C01779=-54.382,79.482,17.095,174.9324,20.6601,-3295.6199
C01780=-53.070,81.058,17.237,173.5629,15.1731,-3296.7866
C01781=-52.143,82.495,17.374,174.7815,10.0525,-3297.7041
C01782=-51.202,83.948,17.473,177.1153,6.7838,-3298.6199
C01783=-49.816,85.535,17.521,178.9354,4.2497,-3299.7833
C01784=-47.692,87.339,17.545,179.7213,1.8693,-3301.3630
C01785=-45.077,89.109,17.565,179.9709,0.3614,-3303.1668
C01786=-42.311,90.585,17.585,-179.9996,0.0820,-3304.9634
C01787=-39.610,91.818,17.598,179.9970,0.0075,-3306.6648
C01788=-36.917,92.934,17.598,179.9968,0.0074,-3308.3351
C01789=-34.135,93.972,17.585,179.9985,0.0798,-3310.0366
C01790=-31.135,94.884,17.565,-179.9727,0.3589,-3311.8334
C01791=-28.035,95.481,17.545,-179.7194,1.8706,-3313.6368
C01792=-25.257,95.708,17.521,-178.9370,4.2461,-3315.2169
C01793=-23.155,95.565,17.473,-177.1151,6.7819,-3316.3800
C01794=-21.462,95.203,17.374,-174.7852,10.0480,-3317.2959
C01795=-19.790,94.842,17.237,-173.5645,15.1715,-3318.2136
C01796=-17.748,94.656,17.095,-174.9374,20.6589,-3319.3803
C01797=-14.774,94.777,16.986,-178.0146,24.0591,-3321.1399
C01798=-10.339,95.219,16.941,-179.6989,25.0665,-3323.8030
C01799=-5.406,95.617,16.939,179.9726,25.1250,-3326.7641
C01800=0.000,94.804,18.916,-180.0000,27.0775,-3330.0000
C01801=5.317,94.652,18.914,-179.9702,27.0874,-3333.2152
C01802=10.190,94.262,18.917,179.5911,27.0185,-3336.1699
C01803=14.592,93.857,18.976,177.3137,25.8724,-3338.8371
C01804=17.528,93.824,19.120,173.2655,21.6484,-3340.5819
C01805=19.540,94.146,19.309,171.9611,14.9094,-3341.7253
C01806=21.192,94.676,19.493,173.8561,9.2462,-3342.6169
C01807=22.867,95.222,19.627,176.6046,6.2189,-3343.5035
C01808=24.945,95.538,19.692,178.7208,4.0294,-3344.6333
C01809=27.741,95.446,19.726,179.6779,1.7445,-3346.2063
C01810=30.903,94.927,19.753,179.9766,0.2756,-3348.0324
C01811=33.988,94.020,19.780,179.9962,0.0778,-3349.8748
C01812=36.867,92.953,19.798,-179.9968,0.0074,-3351.6343
C01813=39.659,91.796,19.798,-179.9970,0.0075,-3353.3660
C01814=42.449,90.515,19.780,-179.9981,0.0768,-3355.1253
C01815=45.272,88.975,19.753,-179.9712,0.2718,-3356.9678
C01816=47.874,87.106,19.726,-179.6780,1.7463,-3358.7935
C01817=49.917,85.194,19.692,-178.7206,4.0258,-3360.3670
C01818=51.163,83.502,19.627,-176.6033,6.2165,-3361.4965
C01819=51.961,81.931,19.493,-173.8545,9.2440,-3362.3830
C01820=52.755,80.388,19.309,-171.9613,14.9062,-3363.2751
C01821=53.950,78.738,19.120,-173.2660,21.6521,-3364.4183
C01822=56.048,76.685,18.976,-177.3146,25.8712,-3366.1625
C01823=59.448,73.859,18.917,-179.5906,27.0203,-3368.8301
C01824=63.169,70.689,18.914,179.9644,27.0876,-3371.7846
C01825=67.036,67.036,18.916,-180.0000,27.0793,-3375.0000
C01826=70.689,63.169,18.914,-179.9644,27.0876,-3378.2154
C01827=73.859,59.448,18.917,179.5906,27.0203,-3381.1699
C01828=76.685,56.048,18.976,177.3146,25.8712,-3383.8375
C01829=78.738,53.950,19.120,173.2660,21.6521,-3385.5817
C01830=80.388,52.755,19.309,171.9613,14.9062,-3386.7249
C01831=81.931,51.961,19.493,173.8545,9.2440,-3387.6170
C01832=83.502,51.163,19.627,176.6033,6.2165,-3388.5035
C01833=85.194,49.917,19.692,178.7206,4.0258,-3389.6330
C01834=87.106,47.874,19.726,179.6780,1.7463,-3391.2065
C01835=88.975,45.272,19.753,179.9712,0.2718,-3393.0322
C01836=90.515,42.449,19.780,179.9981,0.0768,-3394.8747
C01837=91.796,39.659,19.798,179.9970,0.0075,-3396.6340
C01838=92.953,36.867,19.798,179.9968,0.0074,-3398.3657
C01839=94.020,33.988,19.780,-179.9962,0.0778,-3400.1252
C01840=94.927,30.903,19.753,-179.9766,0.2756,-3401.9676
C01841=95.446,27.741,19.726,-179.6779,1.7445,-3403.7937
C01842=95.538,24.945,19.692,-178.7208,4.0294,-3405.3667
C01843=95.222,22.867,19.627,-176.6046,6.2189,-3406.4965
C01844=94.676,21.192,19.493,-173.8561,9.2462,-3407.3831
C01845=94.146,19.540,19.309,-171.9611,14.9094,-3408.2747
C01846=93.824,17.528,19.120,-173.2655,21.6484,-3409.4181
C01847=93.857,14.592,18.976,-177.3137,25.8724,-3411.1629
C01848=94.262,10.190,18.917,-179.5911,27.0185,-3413.8301
C01849=94.652,5.317,18.914,179.9702,27.0874,-3416.7848
C01850=94.804,0.000,18.916,180.0000,27.0775,-3420.0000
C01851=94.652,-5.317,18.914,-179.9702,27.0874,-3423.2152
C01852=94.262,-10.190,18.917,179.5911,27.0185,-3426.1699
C01853=93.857,-14.592,18.976,177.3137,25.8724,-3428.8371
C01854=93.824,-17.528,19.120,173.2655,21.6484,-3430.5819
C01855=94.146,-19.540,19.309,171.9611,14.9094,-3431.7253
C01856=94.676,-21.192,19.493,173.8561,9.2462,-3432.6169
C01857=95.222,-22.867,19.627,176.6046,6.2189,-3433.5035
C01858=95.538,-24.945,19.692,178.7208,4.0294,-3434.6333
C01859=95.446,-27.741,19.726,179.6779,1.7445,-3436.2063
C01860=94.927,-30.903,19.753,179.9766,0.2756,-3438.0324
C01861=94.020,-33.988,19.780,179.9962,0.0778,-3439.8748
C01862=92.953,-36.867,19.798,-179.9968,0.0074,-3441.6343
C01863=91.796,-39.659,19.798,-179.9970,0.0075,-3443.3660
C01864=90.515,-42.449,19.780,-179.9981,0.0768,-3445.1253
C01865=88.975,-45.272,19.753,-179.9712,0.2718,-3446.9678
C01866=87.106,-47.874,19.726,-179.6780,1.7463,-3448.7935
C01867=85.194,-49.917,19.692,-178.7206,4.0258,-3450.3670
C01868=83.502,-51.163,19.627,-176.6033,6.2165,-3451.4965
C01869=81.931,-51.961,19.493,-173.8545,9.2440,-3452.3830
C01870=80.388,-52.755,19.309,-171.9613,14.9062,-3453.2751
C01871=78.738,-53.950,19.120,-173.2660,21.6521,-3454.4183
C01872=76.685,-56.048,18.976,-177.3146,25.8712,-3456.1625
C01873=73.859,-59.448,18.917,-179.5906,27.0203,-3458.8301
C01874=70.689,-63.169,18.914,179.9644,27.0876,-3461.7846
C01875=67.036,-67.036,18.916,-180.0000,27.0793,-3465.0000
C01876=63.169,-70.689,18.914,-179.9644,27.0876,-3468.2154
C01877=59.448,-73.859,18.917,179.5906,27.0203,-3471.1699
C01878=56.048,-76.685,18.976,177.3146,25.8712,-3473.8375
C01879=53.950,-78.738,19.120,173.2660,21.6521,-3475.5817
C01880=52.755,-80.388,19.309,171.9613,14.9062,-3476.7249
C01881=51.961,-81.931,19.493,173.8545,9.2440,-3477.6170
C01882=51.163,-83.502,19.627,176.6033,6.2165,-3478.5035
C01883=49.917,-85.194,19.692,178.7206,4.0258,-3479.6330
C01884=47.874,-87.106,19.726,179.6780,1.7463,-3481.2065
C01885=45.272,-88.975,19.753,179.9712,0.2718,-3483.0322
C01886=42.449,-90.515,19.780,179.9981,0.0768,-3484.8747
C01887=39.659,-91.796,19.798,179.9970,0.0075,-3486.6340
C01888=36.867,-92.953,19.798,179.9968,0.0074,-3488.3657
C01889=33.988,-94.020,19.780,-179.9962,0.0778,-3490.1252
C01890=30.903,-94.927,19.753,-179.9766,0.2756,-3491.9676
C01891=27.741,-95.446,19.726,-179.6779,1.7445,-3493.7937
C01892=24.945,-95.538,19.692,-178.7208,4.0294,-3495.3667
C01893=22.867,-95.222,19.627,-176.6046,6.2189,-3496.4965
C01894=21.192,-94.676,19.493,-173.8561,9.2462,-3497.3831
C01895=19.540,-94.146,19.309,-171.9611,14.9094,-3498.2747
C01896=17.528,-93.824,19.120,-173.2655,21.6484,-3499.4181
C01897=14.592,-93.857,18.976,-177.3137,25.8724,-3501.1629
C01898=10.190,-94.262,18.917,-179.5911,27.0185,-3503.8301
C01899=5.317,-94.652,18.914,179.9702,27.0874,-3506.7848
C01900=0.000,-94.804,18.916,-180.0000,27.0775,-3510.0000
C01901=-5.317,-94.652,18.914,-179.9702,27.0874,-3513.2152
C01902=-10.190,-94.262,18.917,179.5911,27.0185,-3516.1699
C01903=-14.592,-93.857,18.976,177.3137,25.8724,-3518.8371
C01904=-17.528,-93.824,19.120,173.2655,21.6484,-3520.5819
C01905=-19.540,-94.146,19.309,171.9611,14.9094,-3521.7253
C01906=-21.192,-94.676,19.493,173.8561,9.2462,-3522.6169
C01907=-22.867,-95.222,19.627,176.6046,6.2189,-3523.5035
C01908=-24.945,-95.538,19.692,178.7208,4.0294,-3524.6333
C01909=-27.741,-95.446,19.726,179.6779,1.7445,-3526.2063
C01910=-30.903,-94.927,19.753,179.9766,0.2756,-3528.0324
C01911=-33.988,-94.020,19.780,179.9962,0.0778,-3529.8748
C01912=-36.867,-92.953,19.798,-179.9968,0.0074,-3531.6343
C01913=-39.659,-91.796,19.798,-179.9970,0.0075,-3533.3660
C01914=-42.449,-90.515,19.780,-179.9981,0.0768,-3535.1253
C01915=-45.272,-88.975,19.753,-179.9712,0.2718,-3536.9678
C01916=-47.874,-87.106,19.726,-179.6780,1.7463,-3538.7935
C01917=-49.917,-85.194,19.692,-178.7206,4.0258,-3540.3670
C01918=-51.163,-83.502,19.627,-176.6033,6.2165,-3541.4965
C01919=-51.961,-81.931,19.493,-173.8545,9.2440,-3542.3830
C01920=-52.755,-80.388,19.309,-171.9613,14.9062,-3543.2751
C01921=-53.950,-78.738,19.120,-173.2660,21.6521,-3544.4183
C01922=-56.048,-76.685,18.976,-177.3146,25.8712,-3546.1625
C01923=-59.448,-73.859,18.917,-179.5906,27.0203,-3548.8301
C01924=-63.169,-70.689,18.914,179.9644,27.0876,-3551.7846
C01925=-67.036,-67.036,18.916,180.0000,27.0793,-3555.0000
C01926=-70.689,-63.169,18.914,-179.9644,27.0876,-3558.2154
C01927=-73.859,-59.448,18.917,179.5906,27.0203,-3561.1699
C01928=-76.685,-56.048,18.976,177.3146,25.8712,-3563.8375
C01929=-78.738,-53.950,19.120,173.2660,21.6521,-3565.5817
C01930=-80.388,-52.755,19.309,171.9613,14.9062,-3566.7249
C01931=-81.931,-51.961,19.493,173.8545,9.2440,-3567.6170
C01932=-83.502,-51.163,19.627,176.6033,6.2165,-3568.5035
C01933=-85.194,-49.917,19.692,178.7206,4.0258,-3569.6330
C01934=-87.106,-47.874,19.726,179.6780,1.7463,-3571.2065
C01935=-88.975,-45.272,19.753,179.9712,0.2718,-3573.0322
C01936=-90.515,-42.449,19.780,179.9981,0.0768,-3574.8747
C01937=-91.796,-39.659,19.798,179.9970,0.0075,-3576.6340
C01938=-92.953,-36.867,19.798,179.9968,0.0074,-3578.3657
C01939=-94.020,-33.988,19.780,-179.9962,0.0778,-3580.1252
C01940=-94.927,-30.903,19.753,-179.9766,0.2756,-3581.9676
C01941=-95.446,-27.741,19.726,-179.6779,1.7445,-3583.7937
C01942=-95.538,-24.945,19.692,-178.7208,4.0294,-3585.3667
C01943=-95.222,-22.867,19.627,-176.6046,6.2189,-3586.4965
C01944=-94.676,-21.192,19.493,-173.8561,9.2462,-3587.3831
C01945=-94.146,-19.540,19.309,-171.9611,14.9094,-3588.2747
C01946=-93.824,-17.528,19.120,-173.2655,21.6484,-3589.4181
C01947=-93.857,-14.592,18.976,-177.3137,25.8724,-3591.1629
C01948=-94.262,-10.190,18.917,-179.5911,27.0185,-3593.8301
C01949=-94.652,-5.317,18.914,179.9702,27.0874,-3596.7848
C01950=-94.804,0.000,18.916,-180.0000,27.0775,-3600.0000
C01951=-94.652,5.317,18.914,-179.9702,27.0874,-3603.2152
C01952=-94.262,10.190,18.917,179.5911,27.0185,-3606.1699
C01953=-93.857,14.592,18.976,177.3137,25.8724,-3608.8371
C01954=-93.824,17.528,19.120,173.2655,21.6484,-3610.5819
C01955=-94.146,19.540,19.309,171.9611,14.9094,-3611.7253
C01956=-94.676,21.192,19.493,173.8561,9.2462,-3612.6169
C01957=-95.222,22.867,19.627,176.6046,6.2189,-3613.5035
C01958=-95.538,24.945,19.692,178.7208,4.0294,-3614.6333
C01959=-95.446,27.741,19.726,179.6779,1.7445,-3616.2063
C01960=-94.927,30.903,19.753,179.9766,0.2756,-3618.0324
C01961=-94.020,33.988,19.780,179.9962,0.0778,-3619.8748
C01962=-92.953,36.867,19.798,-179.9968,0.0074,-3621.6343
C01963=-91.796,39.659,19.798,-179.9970,0.0075,-3623.3660
C01964=-90.515,42.449,19.780,-179.9981,0.0768,-3625.1253
C01965=-88.975,45.272,19.753,-179.9712,0.2718,-3626.9678
C01966=-87.106,47.874,19.726,-179.6780,1.7463,-3628.7935
C01967=-85.194,49.917,19.692,-178.7206,4.0258,-3630.3670
C01968=-83.502,51.163,19.627,-176.6033,6.2165,-3631.4965
C01969=-81.931,51.961,19.493,-173.8545,9.2440,-3632.3830
C01970=-80.388,52.755,19.309,-171.9613,14.9062,-3633.2751
C01971=-78.738,53.950,19.120,-173.2660,21.6521,-3634.4183
C01972=-76.685,56.048,18.976,-177.3146,25.8712,-3636.1625
C01973=-73.859,59.448,18.917,-179.5906,27.0203,-3638.8301
C01974=-70.689,63.169,18.914,179.9644,27.0876,-3641.7846
C01975=-67.036,67.036,18.916,180.0000,27.0793,-3645.0000
C01976=-63.169,70.689,18.914,-179.9644,27.0876,-3648.2154
C01977=-59.448,73.859,18.917,179.5906,27.0203,-3651.1699
C01978=-56.048,76.685,18.976,177.3146,25.8712,-3653.8375
C01979=-53.950,78.738,19.120,173.2660,21.6521,-3655.5817
C01980=-52.755,80.388,19.309,171.9613,14.9062,-3656.7249
C01981=-51.961,81.931,19.493,173.8545,9.2440,-3657.6170
C01982=-51.163,83.502,19.627,176.6033,6.2165,-3658.5035
C01983=-49.917,85.194,19.692,178.7206,4.0258,-3659.6330
C01984=-47.874,87.106,19.726,179.6780,1.7463,-3661.2065
C01985=-45.272,88.975,19.753,179.9712,0.2718,-3663.0322
C01986=-42.449,90.515,19.780,179.9981,0.0768,-3664.8747
C01987=-39.659,91.796,19.798,179.9970,0.0075,-3666.6340
C01988=-36.867,92.953,19.798,179.9968,0.0074,-3668.3657
C01989=-33.988,94.020,19.780,-179.9962,0.0778,-3670.1252
C01990=-30.903,94.927,19.753,-179.9766,0.2756,-3671.9676
C01991=-27.741,95.446,19.726,-179.6779,1.7445,-3673.7937
C01992=-24.945,95.538,19.692,-178.7208,4.0294,-3675.3667
C01993=-22.867,95.222,19.627,-176.6046,6.2189,-3676.4965
C01994=-21.192,94.676,19.493,-173.8561,9.2462,-3677.3831
C01995=-19.540,94.146,19.309,-171.9611,14.9094,-3678.2747
C01996=-17.528,93.824,19.120,-173.2655,21.6484,-3679.4181
C01997=-14.592,93.857,18.976,-177.3137,25.8724,-3681.1629
C01998=-10.190,94.262,18.917,-179.5911,27.0185,-3683.8301
C01999=-5.317,94.652,18.914,179.9702,27.0874,-3686.7848
///TOOL 0
///POSTYPE ANGLE
///ANGLE
EC00000=0.0000,90.0000
EC00001=0.0000,93.3204
EC00002=0.0000,96.3084
EC00003=0.0000,98.9540
EC00004=0.0000,100.7765
EC00005=0.0000,102.0369
EC00006=0.0000,103.0576
EC00007=0.0000,104.0938
EC00008=0.0000,105.3967
EC00009=0.0000,107.0065
EC00010=0.0000,108.7198
EC00011=0.0000,110.3278
EC00012=0.0000,111.7902
EC00013=0.0000,113.2098
EC00014=0.0000,114.6724
EC00015=-0.0000,116.2801
EC00016=-0.0000,117.9935
EC00017=0.0000,119.6039
EC00018=0.0000,120.9060
EC00019=0.0000,121.9421
EC00020=0.0000,122.9632
EC00021=0.0000,124.2234
EC00022=0.0000,126.0464
EC00023=0.0000,128.6909
EC00024=0.0000,131.6796
EC00025=0.0000,135.0000
EC00026=0.0000,138.3204
EC00027=0.0000,141.3091
EC00028=-0.0000,143.9536
EC00029=0.0000,145.7766
EC00030=0.0000,147.0368
EC00031=0.0000,148.0579
EC00032=0.0000,149.0940
EC00033=0.0000,150.3961
EC00034=0.0000,152.0065
EC00035=0.0000,153.7199
EC00036=0.0000,155.3276
EC00037=0.0000,156.7902
EC00038=0.0000,158.2098
EC00039=0.0000,159.6722
EC00040=0.0000,161.2802
EC00041=0.0000,162.9935
EC00042=0.0000,164.6033
EC00043=0.0000,165.9062
EC00044=0.0000,166.9424
EC00045=0.0000,167.9631
EC00046=0.0000,169.2235
EC00047=0.0000,171.0460
EC00048=0.0000,173.6916
EC00049=0.0000,176.6796
EC00050=0.0000,180.0000
EC00051=0.0000,183.3204
EC00052=0.0000,186.3084
EC00053=0.0000,188.9540
EC00054=0.0000,190.7765
EC00055=0.0000,192.0369
EC00056=0.0000,193.0576
EC00057=0.0000,194.0938
EC00058=0.0000,195.3967
EC00059=0.0000,197.0065
EC00060=0.0000,198.7198
EC00061=0.0000,200.3278
EC00062=0.0000,201.7902
EC00063=0.0000,203.2098
EC00064=0.0000,204.6724
EC00065=0.0000,206.2801
EC00066=0.0000,207.9935
EC00067=0.0000,209.6039
EC00068=0.0000,210.9060
EC00069=0.0000,211.9421
EC00070=0.0000,212.9632
EC00071=0.0000,214.2234
EC00072=0.0000,216.0464
EC00073=0.0000,218.6909
EC00074=0.0000,221.6796
EC00075=0.0000,225.0000
EC00076=0.0000,228.3204
EC00077=0.0000,231.3091
EC00078=0.0000,233.9536
EC00079=0.0000,235.7766
EC00080=0.0000,237.0368
EC00081=0.0000,238.0579
EC00082=0.0000,239.0940
EC00083=-0.0000,240.3961
EC00084=0.0000,242.0065
EC00085=0.0000,243.7199
EC00086=0.0000,245.3276
EC00087=0.0000,246.7902
EC00088=0.0000,248.2098
EC00089=0.0000,249.6722
EC00090=0.0000,251.2802
EC00091=0.0000,252.9935
EC00092=0.0000,254.6033
EC00093=0.0000,255.9062
EC00094=0.0000,256.9424
EC00095=0.0000,257.9631
EC00096=0.0000,259.2235
EC00097=0.0000,261.0460
EC00098=0.0000,263.6916
EC00099=0.0000,266.6796
EC00100=-0.0000,270.0000
EC00101=-0.0000,273.3204
EC00102=-0.0000,276.3084
EC00103=-0.0000,278.9540
EC00104=-0.0000,280.7765
EC00105=-0.0000,282.0369
EC00106=-0.0000,283.0576
EC00107=-0.0000,284.0938
EC00108=-0.0000,285.3967
EC00109=-0.0000,287.0065
EC00110=-0.0000,288.7198
EC00111=-0.0000,290.3278
EC00112=-0.0000,291.7902
EC00113=-0.0000,293.2098
EC00114=-0.0000,294.6724
EC00115=-0.0000,296.2801
EC00116=-0.0000,297.9935
EC00117=-0.0000,299.6039
EC00118=-0.0000,300.9060
EC00119=-0.0000,301.9421
EC00120=-0.0000,302.9632
EC00121=-0.0000,304.2234
EC00122=-0.0000,306.0464
EC00123=-0.0000,308.6909
EC00124=-0.0000,311.6796
EC00125=-0.0000,315.0000
EC00126=-0.0000,318.3204
EC00127=-0.0000,321.3091
EC00128=-0.0000,323.9536
EC00129=-0.0000,325.7766
EC00130=-0.0000,327.0368
EC00131=-0.0000,328.0579
EC00132=-0.0000,329.0940
EC00133=-0.0000,330.3961
EC00134=-0.0000,332.0065
EC00135=-0.0000,333.7199
EC00136=0.0000,335.3276
EC00137=0.0000,336.7902
EC00138=-0.0000,338.2098
EC00139=-0.0000,339.6722
EC00140=0.0000,341.2802
EC00141=0.0000,342.9935
EC00142=-0.0000,344.6033
EC00143=-0.0000,345.9062
EC00144=-0.0000,346.9424
EC00145=-0.0000,347.9631
EC00146=-0.0000,349.2235
EC00147=-0.0000,351.0460
EC00148=-0.0000,353.6916
EC00149=-0.0000,356.6796
EC00150=0.0000,360.0000
EC00151=0.0000,363.3204
EC00152=0.0000,366.3084
EC00153=0.0000,368.9540
EC00154=0.0000,370.7765
EC00155=0.0000,372.0369
EC00156=0.0000,373.0576
EC00157=0.0000,374.0938
EC00158=0.0000,375.3967
EC00159=0.0000,377.0065
EC00160=0.0000,378.7198
EC00161=0.0000,380.3278
EC00162=0.0000,381.7902
EC00163=0.0000,383.2098
EC00164=0.0000,384.6724
EC00165=0.0000,386.2801
EC00166=0.0000,387.9935
EC00167=0.0000,389.6039
EC00168=0.0000,390.9060
EC00169=0.0000,391.9421
EC00170=0.0000,392.9632
EC00171=0.0000,394.2234
EC00172=0.0000,396.0464
EC00173=0.0000,398.6909
EC00174=0.0000,401.6796
EC00175=0.0000,405.0000
EC00176=0.0000,408.3204
EC00177=0.0000,411.3091
EC00178=0.0000,413.9536
EC00179=0.0000,415.7766
EC00180=0.0000,417.0368
EC00181=0.0000,418.0579
EC00182=0.0000,419.0940
EC00183=0.0000,420.3961
EC00184=0.0000,422.0065
EC00185=0.0000,423.7199
EC00186=0.0000,425.3276
EC00187=0.0000,426.7902
EC00188=0.0000,428.2098
EC00189=0.0000,429.6722
EC00190=0.0000,431.2802
EC00191=0.0000,432.9935
EC00192=0.0000,434.6033
EC00193=0.0000,435.9062
EC00194=0.0000,436.9424
EC00195=0.0000,437.9631
EC00196=0.0000,439.2235
EC00197=0.0000,441.0460
EC00198=0.0000,443.6916
EC00199=0.0000,446.6796
EC00200=4.0599,450.0000
EC00201=4.0610,453.3190
EC00202=4.0560,456.3064
EC00203=3.8999,458.9521
EC00204=3.4994,460.7740
EC00205=2.9093,462.0325
EC00206=2.2192,463.0515
EC00207=1.5274,464.0856
EC00208=0.9256,465.3858
EC00209=0.4495,466.9948
EC00210=0.1268,468.7100
EC00211=0.0181,470.3211
EC00212=0.0000,471.7884
EC00213=0.0000,473.2118
EC00214=0.0204,474.6788
EC00215=0.1281,476.2904
EC00216=0.4486,478.0051
EC00217=0.9267,479.6142
EC00218=1.5272,480.9142
EC00219=2.2211,481.9485
EC00220=2.9093,482.9671
EC00221=3.4970,484.2260
EC00222=3.8982,486.0482
EC00223=4.0551,488.6933
EC00224=4.0616,491.6811
EC00225=4.0629,495.0000
EC00226=4.0616,498.3189
EC00227=4.0551,501.3067
EC00228=3.8982,503.9518
EC00229=3.4970,505.7740
EC00230=2.9093,507.0329
EC00231=2.2211,508.0515
EC00232=1.5272,509.0858
EC00233=0.9267,510.3858
EC00234=0.4486,511.9949
EC00235=0.1281,513.7096
EC00236=0.0204,515.3212
EC00237=0.0000,516.7882
EC00238=0.0000,518.2116
EC00239=0.0181,519.6789
EC00240=0.1268,521.2900
EC00241=0.4495,523.0052
EC00242=0.9256,524.6142
EC00243=1.5274,525.9144
EC00244=2.2192,526.9485
EC00245=2.9093,527.9675
EC00246=3.4994,529.2260
EC00247=3.8999,531.0479
EC00248=4.0560,533.6936
EC00249=4.0610,536.6810
EC00250=4.0599,540.0000
EC00251=4.0610,543.3190
EC00252=4.0560,546.3064
EC00253=3.8999,548.9521
EC00254=3.4994,550.7740
EC00255=2.9093,552.0325
EC00256=2.2192,553.0515
EC00257=1.5274,554.0856
EC00258=0.9256,555.3858
EC00259=0.4495,556.9948
EC00260=0.1268,558.7100
EC00261=0.0181,560.3211
EC00262=0.0000,561.7884
EC00263=0.0000,563.2118
EC00264=0.0204,564.6788
EC00265=0.1281,566.2904
EC00266=0.4486,568.0051
EC00267=0.9267,569.6142
EC00268=1.5272,570.9142
EC00269=2.2211,571.9485
EC00270=2.9093,572.9671
EC00271=3.4970,574.2260
EC00272=3.8982,576.0482
EC00273=4.0551,578.6933
EC00274=4.0616,581.6811
EC00275=4.0629,585.0000
EC00276=4.0616,588.3189
EC00277=4.0551,591.3067
EC00278=3.8982,593.9518
EC00279=3.4970,595.7740
EC00280=2.9093,597.0329
EC00281=2.2211,598.0515
EC00282=1.5272,599.0858
EC00283=0.9267,600.3858
EC00284=0.4486,601.9949
EC00285=0.1281,603.7096
EC00286=0.0204,605.3212
EC00287=0.0000,606.7882
EC00288=0.0000,608.2116
EC00289=0.0181,609.6789
EC00290=0.1268,611.2900
EC00291=0.4495,613.0052
EC00292=0.9256,614.6142
EC00293=1.5274,615.9144
EC00294=2.2192,616.9485
EC00295=2.9093,617.9675
EC00296=3.4994,619.2260
EC00297=3.8999,621.0479
EC00298=4.0560,623.6936
EC00299=4.0610,626.6810
EC00300=4.0599,630.0000
EC00301=4.0610,633.3190
EC00302=4.0560,636.3064
EC00303=3.8999,638.9521
EC00304=3.4994,640.7740
EC00305=2.9093,642.0325
EC00306=2.2192,643.0515
EC00307=1.5274,644.0856
EC00308=0.9256,645.3858
EC00309=0.4495,646.9948
EC00310=0.1268,648.7100
EC00311=0.0181,650.3211
EC00312=0.0000,651.7884
EC00313=0.0000,653.2118
EC00314=0.0204,654.6788
EC00315=0.1281,656.2904
EC00316=0.4486,658.0051
EC00317=0.9267,659.6142
EC00318=1.5272,660.9142
EC00319=2.2211,661.9485
EC00320=2.9093,662.9671
EC00321=3.4970,664.2260
EC00322=3.8982,666.0482
EC00323=4.0551,668.6933
EC00324=4.0616,671.6811
EC00325=4.0629,675.0000
EC00326=4.0616,678.3189
EC00327=4.0551,681.3067
EC00328=3.8982,683.9518
EC00329=3.4970,685.7740
EC00330=2.9093,687.0329
EC00331=2.2211,688.0515
EC00332=1.5272,689.0858
EC00333=0.9267,690.3858
EC00334=0.4486,691.9949
EC00335=0.1281,693.7096
EC00336=0.0204,695.3212
EC00337=0.0000,696.7882
EC00338=0.0000,698.2116
EC00339=0.0181,699.6789
EC00340=0.1268,701.2900
EC00341=0.4495,703.0052
EC00342=0.9256,704.6142
EC00343=1.5274,705.9144
EC00344=2.2192,706.9485
EC00345=2.9093,707.9675
EC00346=3.4994,709.2260
EC00347=3.8999,711.0479
EC00348=4.0560,713.6936
EC00349=4.0610,716.6810
EC00350=4.0599,720.0000
EC00351=4.0610,723.3190
EC00352=4.0560,726.3064
EC00353=3.8999,728.9521
EC00354=3.4994,730.7740
EC00355=2.9093,732.0325
EC00356=2.2192,733.0515
EC00357=1.5274,734.0856
EC00358=0.9256,735.3858
EC00359=0.4495,736.9948
EC00360=0.1268,738.7100
EC00361=0.0181,740.3211
EC00362=0.0000,741.7884
EC00363=0.0000,743.2118
EC00364=0.0204,744.6788
EC00365=0.1281,746.2904
EC00366=0.4486,748.0051
EC00367=0.9267,749.6142
EC00368=1.5272,750.9142
EC00369=2.2211,751.9485
EC00370=2.9093,752.9671
EC00371=3.4970,754.2260
EC00372=3.8982,756.0482
EC00373=4.0551,758.6933
EC00374=4.0616,761.6811
EC00375=4.0629,765.0000
EC00376=4.0616,768.3189
EC00377=4.0551,771.3067
EC00378=3.8982,773.9518
EC00379=3.4970,775.7740
EC00380=2.9093,777.0329
EC00381=2.2211,778.0515
EC00382=1.5272,779.0858
EC00383=0.9267,780.3858
EC00384=0.4486,781.9949
EC00385=0.1281,783.7096
EC00386=0.0204,785.3212
EC00387=0.0000,786.7882
EC00388=0.0000,788.2116
EC00389=0.0181,789.6789
EC00390=0.1268,791.2900
EC00391=0.4495,793.0052
EC00392=0.9256,794.6142
EC00393=1.5274,795.9144
EC00394=2.2192,796.9485
EC00395=2.9093,797.9675
EC00396=3.4994,799.2260
EC00397=3.8999,801.0479
EC00398=4.0560,803.6936
EC00399=4.0610,806.6810
EC00400=7.8975,810.0000
EC00401=7.8994,813.3146
EC00402=7.8868,816.3008
EC00403=7.5851,818.9471
EC00404=6.8083,820.7659
EC00405=5.6544,822.0199
EC00406=4.3065,823.0335
EC00407=2.9528,824.0616
EC00408=1.7872,825.3544
EC00409=0.8539,826.9622
EC00410=0.2410,828.6812
EC00411=0.0362,830.3024
EC00412=0.0053,831.7817
EC00413=0.0053,833.2185
EC00414=0.0384,834.6975
EC00415=0.2434,836.3188
EC00416=0.8564,838.0383
EC00417=1.7904,839.6456
EC00418=2.9520,840.9386
EC00419=4.3050,841.9667
EC00420=5.6572,842.9801
EC00421=6.8088,844.2340
EC00422=7.5869,846.0529
EC00423=7.8870,848.6992
EC00424=7.9022,851.6856
EC00425=7.9010,855.0000
EC00426=7.9022,858.3144
EC00427=7.8870,861.3008
EC00428=7.5869,863.9471
EC00429=6.8088,865.7660
EC00430=5.6572,867.0199
EC00431=4.3050,868.0333
EC00432=2.9520,869.0614
EC00433=1.7904,870.3544
EC00434=0.8564,871.9617
EC00435=0.2434,873.6812
EC00436=0.0384,875.3025
EC00437=0.0053,876.7815
EC00438=0.0053,878.2183
EC00439=0.0362,879.6976
EC00440=0.2410,881.3188
EC00441=0.8539,883.0378
EC00442=1.7872,884.6456
EC00443=2.9528,885.9384
EC00444=4.3065,886.9665
EC00445=5.6544,887.9801
EC00446=6.8083,889.2341
EC00447=7.5851,891.0529
EC00448=7.8868,893.6992
EC00449=7.8994,896.6854
EC00450=7.8975,900.0000
EC00451=7.8994,903.3146
EC00452=7.8868,906.3008
EC00453=7.5851,908.9471
EC00454=6.8083,910.7659
EC00455=5.6544,912.0199
EC00456=4.3065,913.0335
EC00457=2.9528,914.0616
EC00458=1.7872,915.3544
EC00459=0.8539,916.9622
EC00460=0.2410,918.6812
EC00461=0.0362,920.3024
EC00462=0.0053,921.7817
EC00463=0.0053,923.2185
EC00464=0.0384,924.6975
EC00465=0.2434,926.3188
EC00466=0.8564,928.0383
EC00467=1.7904,929.6456
EC00468=2.9520,930.9386
EC00469=4.3050,931.9667
EC00470=5.6572,932.9801
EC00471=6.8088,934.2340
EC00472=7.5869,936.0529
EC00473=7.8870,938.6992
EC00474=7.9022,941.6856
EC00475=7.9010,945.0000
EC00476=7.9022,948.3144
EC00477=7.8870,951.3008
EC00478=7.5869,953.9471
EC00479=6.8088,955.7660
EC00480=5.6572,957.0199
EC00481=4.3050,958.0333
EC00482=2.9520,959.0614
EC00483=1.7904,960.3544
EC00484=0.8564,961.9617
EC00485=0.2434,963.6812
EC00486=0.0384,965.3025
EC00487=0.0053,966.7815
EC00488=0.0053,968.2183
EC00489=0.0362,969.6976
EC00490=0.2410,971.3188
EC00491=0.8539,973.0378
EC00492=1.7872,974.6456
EC00493=2.9528,975.9384
EC00494=4.3065,976.9665
EC00495=5.6544,977.9801
EC00496=6.8083,979.2341
EC00497=7.5851,981.0529
EC00498=7.8868,983.6992
EC00499=7.8994,986.6854
EC00500=7.8975,990.0000
EC00501=7.8994,993.3146
EC00502=7.8868,996.3008
EC00503=7.5851,998.9471
EC00504=6.8083,1000.7659
EC00505=5.6544,1002.0199
EC00506=4.3065,1003.0335
EC00507=2.9528,1004.0616
EC00508=1.7872,1005.3544
EC00509=0.8539,1006.9622
EC00510=0.2410,1008.6812
EC00511=0.0362,1010.3024
EC00512=0.0053,1011.7817
EC00513=0.0053,1013.2185
EC00514=0.0384,1014.6975
EC00515=0.2434,1016.3188
EC00516=0.8564,1018.0383
EC00517=1.7904,1019.6456
EC00518=2.9520,1020.9386
EC00519=4.3050,1021.9667
EC00520=5.6572,1022.9801
EC00521=6.8088,1024.2340
EC00522=7.5869,1026.0529
EC00523=7.8870,1028.6992
EC00524=7.9022,1031.6856
EC00525=7.9010,1035.0000
EC00526=7.9022,1038.3144
EC00527=7.8870,1041.3008
EC00528=7.5869,1043.9471
EC00529=6.8088,1045.7660
EC00530=5.6572,1047.0199
EC00531=4.3050,1048.0333
EC00532=2.9520,1049.0614
EC00533=1.7904,1050.3544
EC00534=0.8564,1051.9617
EC00535=0.2434,1053.6812
EC00536=0.0384,1055.3025
EC00537=0.0053,1056.7815
EC00538=0.0053,1058.2183
EC00539=0.0362,1059.6976
EC00540=0.2410,1061.3188
EC00541=0.8539,1063.0378
EC00542=1.7872,1064.6456
EC00543=2.9528,1065.9384
EC00544=4.3065,1066.9665
EC00545=5.6544,1067.9801
EC00546=6.8083,1069.2341
EC00547=7.5851,1071.0529
EC00548=7.8868,1073.6992
EC00549=7.8994,1076.6854
EC00550=7.8975,1080.0000
EC00551=7.8994,1083.3146
EC00552=7.8868,1086.3008
EC00553=7.5851,1088.9471
EC00554=6.8083,1090.7659
EC00555=5.6544,1092.0199
EC00556=4.3065,1093.0335
EC00557=2.9528,1094.0616
EC00558=1.7872,1095.3544
EC00559=0.8539,1096.9622
EC00560=0.2410,1098.6812
EC00561=0.0362,1100.3024
EC00562=0.0053,1101.7817
EC00563=0.0053,1103.2185
EC00564=0.0384,1104.6975
EC00565=0.2434,1106.3188
EC00566=0.8564,1108.0383
EC00567=1.7904,1109.6456
EC00568=2.9520,1110.9386
EC00569=4.3050,1111.9667
EC00570=5.6572,1112.9801
EC00571=6.8088,1114.2340
EC00572=7.5869,1116.0529
EC00573=7.8870,1118.6992
EC00574=7.9022,1121.6856
EC00575=7.9010,1125.0000
EC00576=7.9022,1128.3144
EC00577=7.8870,1131.3008
EC00578=7.5869,1133.9471
EC00579=6.8088,1135.7660
EC00580=5.6572,1137.0199
EC00581=4.3050,1138.0333
EC00582=2.9520,1139.0614
EC00583=1.7904,1140.3544
EC00584=0.8564,1141.9617
EC00585=0.2434,1143.6812
EC00586=0.0384,1145.3025
EC00587=0.0053,1146.7815
EC00588=0.0053,1148.2183
EC00589=0.0362,1149.6976
EC00590=0.2410,1151.3188
EC00591=0.8539,1153.0378
EC00592=1.7872,1154.6456
EC00593=2.9528,1155.9384
EC00594=4.3065,1156.9665
EC00595=5.6544,1157.9801
EC00596=6.8083,1159.2341
EC00597=7.5851,1161.0529
EC00598=7.8868,1163.6992
EC00599=7.8994,1166.6854
EC00600=11.4729,1170.0000
EC00601=11.4747,1173.3073
EC00602=11.4524,1176.2913
EC00603=11.0220,1178.9391
EC00604=9.8830,1180.7524
EC00605=8.1850,1181.9986
EC00606=6.1969,1183.0036
EC00607=4.2352,1184.0220
EC00608=2.5536,1185.3030
EC00609=1.2134,1186.9082
EC00610=0.3370,1188.6350
EC00611=0.0543,1190.2716
EC00612=0.0053,1191.7712
EC00613=0.0053,1193.2288
EC00614=0.0564,1194.7282
EC00615=0.3356,1196.3649
EC00616=1.2107,1198.0920
EC00617=2.5592,1199.6973
EC00618=4.2349,1200.9780
EC00619=6.1980,1201.9962
EC00620=8.1891,1203.0013
EC00621=9.8834,1204.2478
EC00622=11.0226,1206.0610
EC00623=11.4500,1208.7088
EC00624=11.4763,1211.6924
EC00625=11.4694,1215.0000
EC00626=11.4763,1218.3076
EC00627=11.4500,1221.2912
EC00628=11.0226,1223.9390
EC00629=9.8834,1225.7522
EC00630=8.1891,1226.9987
EC00631=6.1980,1228.0038
EC00632=4.2349,1229.0220
EC00633=2.5592,1230.3027
EC00634=1.2107,1231.9080
EC00635=0.3356,1233.6351
EC00636=0.0564,1235.2718
EC00637=0.0053,1236.7712
EC00638=0.0053,1238.2288
EC00639=0.0543,1239.7284
EC00640=0.3370,1241.3650
EC00641=1.2134,1243.0918
EC00642=2.5536,1244.6970
EC00643=4.2352,1245.9780
EC00644=6.1969,1246.9964
EC00645=8.1850,1248.0014
EC00646=9.8830,1249.2476
EC00647=11.0220,1251.0609
EC00648=11.4524,1253.7087
EC00649=11.4747,1256.6927
EC00650=11.4729,1260.0000
EC00651=11.4747,1263.3073
EC00652=11.4524,1266.2913
EC00653=11.0220,1268.9391
EC00654=9.8830,1270.7524
EC00655=8.1850,1271.9986
EC00656=6.1969,1273.0036
EC00657=4.2352,1274.0220
EC00658=2.5536,1275.3030
EC00659=1.2134,1276.9082
EC00660=0.3370,1278.6350
EC00661=0.0543,1280.2716
EC00662=0.0053,1281.7712
EC00663=0.0053,1283.2288
EC00664=0.0564,1284.7282
EC00665=0.3356,1286.3649
EC00666=1.2107,1288.0920
EC00667=2.5592,1289.6973
EC00668=4.2349,1290.9780
EC00669=6.1980,1291.9962
EC00670=8.1891,1293.0013
EC00671=9.8834,1294.2478
EC00672=11.0226,1296.0610
EC00673=11.4500,1298.7088
EC00674=11.4763,1301.6924
EC00675=11.4694,1305.0000
EC00676=11.4763,1308.3076
EC00677=11.4500,1311.2912
EC00678=11.0226,1313.9390
EC00679=9.8834,1315.7522
EC00680=8.1891,1316.9987
EC00681=6.1980,1318.0038
EC00682=4.2349,1319.0220
EC00683=2.5592,1320.3027
EC00684=1.2107,1321.9080
EC00685=0.3356,1323.6351
EC00686=0.0564,1325.2718
EC00687=0.0053,1326.7712
EC00688=0.0053,1328.2288
EC00689=0.0543,1329.7284
EC00690=0.3370,1331.3650
EC00691=1.2134,1333.0918
EC00692=2.5536,1334.6970
EC00693=4.2352,1335.9780
EC00694=6.1969,1336.9964
EC00695=8.1850,1338.0014
EC00696=9.8830,1339.2476
EC00697=11.0220,1341.0609
EC00698=11.4524,1343.7087
EC00699=11.4747,1346.6927
EC00700=11.4729,1350.0000
EC00701=11.4747,1353.3073
EC00702=11.4524,1356.2913
EC00703=11.0220,1358.9391
EC00704=9.8830,1360.7524
EC00705=8.1850,1361.9986
EC00706=6.1969,1363.0036
EC00707=4.2352,1364.0220
EC00708=2.5536,1365.3030
EC00709=1.2134,1366.9082
EC00710=0.3370,1368.6350
EC00711=0.0543,1370.2716
EC00712=0.0053,1371.7712
EC00713=0.0053,1373.2288
EC00714=0.0564,1374.7282
EC00715=0.3356,1376.3649
EC00716=1.2107,1378.0920
EC00717=2.5592,1379.6973
EC00718=4.2349,1380.9780
EC00719=6.1980,1381.9962
EC00720=8.1891,1383.0013
EC00721=9.8834,1384.2478
EC00722=11.0226,1386.0610
EC00723=11.4500,1388.7088
EC00724=11.4763,1391.6924
EC00725=11.4694,1395.0000
EC00726=11.4763,1398.3076
EC00727=11.4500,1401.2912
EC00728=11.0226,1403.9390
EC00729=9.8834,1405.7522
EC00730=8.1891,1406.9987
EC00731=6.1980,1408.0038
EC00732=4.2349,1409.0220
EC00733=2.5592,1410.3027
EC00734=1.2107,1411.9080
EC00735=0.3356,1413.6351
EC00736=0.0564,1415.2718
EC00737=0.0053,1416.7712
EC00738=0.0053,1418.2288
EC00739=0.0543,1419.7284
EC00740=0.3370,1421.3650
EC00741=1.2134,1423.0918
EC00742=2.5536,1424.6970
EC00743=4.2352,1425.9780
EC00744=6.1969,1426.9964
EC00745=8.1850,1428.0014
EC00746=9.8830,1429.2476
EC00747=11.0220,1431.0609
EC00748=11.4524,1433.7087
EC00749=11.4747,1436.6927
EC00750=11.4729,1440.0000
EC00751=11.4747,1443.3073
EC00752=11.4524,1446.2913
EC00753=11.0220,1448.9391
EC00754=9.8830,1450.7524
EC00755=8.1850,1451.9986
EC00756=6.1969,1453.0036
EC00757=4.2352,1454.0220
EC00758=2.5536,1455.3030
EC00759=1.2134,1456.9082
EC00760=0.3370,1458.6350
EC00761=0.0543,1460.2716
EC00762=0.0053,1461.7712
EC00763=0.0053,1463.2288
EC00764=0.0564,1464.7282
EC00765=0.3356,1466.3649
EC00766=1.2107,1468.0920
EC00767=2.5592,1469.6973
EC00768=4.2349,1470.9780
EC00769=6.1980,1471.9962
EC00770=8.1891,1473.0013
EC00771=9.8834,1474.2478
EC00772=11.0226,1476.0610
EC00773=11.4500,1478.7088
EC00774=11.4763,1481.6924
EC00775=11.4694,1485.0000
EC00776=11.4763,1488.3076
EC00777=11.4500,1491.2912
EC00778=11.0226,1493.9390
EC00779=9.8834,1495.7522
EC00780=8.1891,1496.9987
EC00781=6.1980,1498.0038
EC00782=4.2349,1499.0220
EC00783=2.5592,1500.3027
EC00784=1.2107,1501.9080
EC00785=0.3356,1503.6351
EC00786=0.0564,1505.2718
EC00787=0.0053,1506.7712
EC00788=0.0053,1508.2288
EC00789=0.0543,1509.7284
EC00790=0.3370,1511.3650
EC00791=1.2134,1513.0918
EC00792=2.5536,1514.6970
EC00793=4.2352,1515.9780
EC00794=6.1969,1516.9964
EC00795=8.1850,1518.0014
EC00796=9.8830,1519.2476
EC00797=11.0220,1521.0609
EC00798=11.4524,1523.7087
EC00799=11.4747,1526.6927
EC00800=14.7616,1530.0000
EC00801=14.7688,1533.2974
EC00802=14.7351,1536.2783
EC00803=14.1865,1538.9284
EC00804=12.6975,1540.7347
EC00805=10.4501,1541.9700
EC00806=7.8426,1542.9633
EC00807=5.3324,1543.9678
EC00808=3.2124,1545.2327
EC00809=1.5081,1546.8342
EC00810=0.4022,1548.5716
EC00811=0.0671,1550.2300
EC00812=0.0074,1551.7565
EC00813=0.0075,1553.2431
EC00814=0.0692,1554.7700
EC00815=0.4023,1556.4284
EC00816=1.5064,1558.1658
EC00817=3.2134,1559.7669
EC00818=5.3325,1561.0323
EC00819=7.8395,1562.0364
EC00820=10.4506,1563.0299
EC00821=12.6950,1564.2655
EC00822=14.1862,1566.0719
EC00823=14.7367,1568.7215
EC00824=14.7681,1571.7023
EC00825=14.7639,1575.0000
EC00826=14.7681,1578.2977
EC00827=14.7367,1581.2785
EC00828=14.1862,1583.9281
EC00829=12.6950,1585.7345
EC00830=10.4506,1586.9701
EC00831=7.8395,1587.9636
EC00832=5.3325,1588.9677
EC00833=3.2134,1590.2331
EC00834=1.5064,1591.8342
EC00835=0.4023,1593.5716
EC00836=0.0692,1595.2300
EC00837=0.0075,1596.7569
EC00838=0.0074,1598.2435
EC00839=0.0671,1599.7700
EC00840=0.4022,1601.4284
EC00841=1.5081,1603.1658
EC00842=3.2124,1604.7673
EC00843=5.3324,1606.0322
EC00844=7.8426,1607.0367
EC00845=10.4501,1608.0300
EC00846=12.6975,1609.2653
EC00847=14.1865,1611.0716
EC00848=14.7351,1613.7217
EC00849=14.7688,1616.7026
EC00850=14.7616,1620.0000
EC00851=14.7688,1623.2974
EC00852=14.7351,1626.2783
EC00853=14.1865,1628.9284
EC00854=12.6975,1630.7347
EC00855=10.4501,1631.9700
EC00856=7.8426,1632.9633
EC00857=5.3324,1633.9678
EC00858=3.2124,1635.2327
EC00859=1.5081,1636.8342
EC00860=0.4022,1638.5716
EC00861=0.0671,1640.2300
EC00862=0.0074,1641.7565
EC00863=0.0075,1643.2431
EC00864=0.0692,1644.7700
EC00865=0.4023,1646.4284
EC00866=1.5064,1648.1658
EC00867=3.2134,1649.7669
EC00868=5.3325,1651.0323
EC00869=7.8395,1652.0364
EC00870=10.4506,1653.0299
EC00871=12.6950,1654.2655
EC00872=14.1862,1656.0719
EC00873=14.7367,1658.7215
EC00874=14.7681,1661.7023
EC00875=14.7639,1665.0000
EC00876=14.7681,1668.2977
EC00877=14.7367,1671.2785
EC00878=14.1862,1673.9281
EC00879=12.6950,1675.7345
EC00880=10.4506,1676.9701
EC00881=7.8395,1677.9636
EC00882=5.3325,1678.9677
EC00883=3.2134,1680.2331
EC00884=1.5064,1681.8342
EC00885=0.4023,1683.5716
EC00886=0.0692,1685.2300
EC00887=0.0075,1686.7569
EC00888=0.0074,1688.2435
EC00889=0.0671,1689.7700
EC00890=0.4022,1691.4284
EC00891=1.5081,1693.1658
EC00892=3.2124,1694.7673
EC00893=5.3324,1696.0322
EC00894=7.8426,1697.0367
EC00895=10.4501,1698.0300
EC00896=12.6975,1699.2653
EC00897=14.1865,1701.0716
EC00898=14.7351,1703.7217
EC00899=14.7688,1706.7026
EC00900=14.7616,1710.0000
EC00901=14.7688,1713.2974
EC00902=14.7351,1716.2783
EC00903=14.1865,1718.9284
EC00904=12.6975,1720.7347
EC00905=10.4501,1721.9700
EC00906=7.8426,1722.9633
EC00907=5.3324,1723.9678
EC00908=3.2124,1725.2327
EC00909=1.5081,1726.8342
EC00910=0.4022,1728.5716
EC00911=0.0671,1730.2300
EC00912=0.0074,1731.7565
EC00913=0.0075,1733.2431
EC00914=0.0692,1734.7700
EC00915=0.4023,1736.4284
EC00916=1.5064,1738.1658
EC00917=3.2134,1739.7669
EC00918=5.3325,1741.0323
EC00919=7.8395,1742.0364
EC00920=10.4506,1743.0299
EC00921=12.6950,1744.2655
EC00922=14.1862,1746.0719
EC00923=14.7367,1748.7215
EC00924=14.7681,1751.7023
EC00925=14.7639,1755.0000
EC00926=14.7681,1758.2977
EC00927=14.7367,1761.2785
EC00928=14.1862,1763.9281
EC00929=12.6950,1765.7345
EC00930=10.4506,1766.9701
EC00931=7.8395,1767.9636
EC00932=5.3325,1768.9677
EC00933=3.2134,1770.2331
EC00934=1.5064,1771.8342
EC00935=0.4023,1773.5716
EC00936=0.0692,1775.2300
EC00937=0.0075,1776.7569
EC00938=0.0074,1778.2435
EC00939=0.0671,1779.7700
EC00940=0.4022,1781.4284
EC00941=1.5081,1783.1658
EC00942=3.2124,1784.7673
EC00943=5.3324,1786.0322
EC00944=7.8426,1787.0367
EC00945=10.4501,1788.0300
EC00946=12.6975,1789.2653
EC00947=14.1865,1791.0716
EC00948=14.7351,1793.7217
EC00949=14.7688,1796.7026
EC00950=14.7616,1800.0000
EC00951=14.7688,1803.2974
EC00952=14.7351,1806.2783
EC00953=14.1865,1808.9284
EC00954=12.6975,1810.7347
EC00955=10.4501,1811.9700
EC00956=7.8426,1812.9633
EC00957=5.3324,1813.9678
EC00958=3.2124,1815.2327
EC00959=1.5081,1816.8342
EC00960=0.4022,1818.5716
EC00961=0.0671,1820.2300
EC00962=0.0074,1821.7565
EC00963=0.0075,1823.2431
EC00964=0.0692,1824.7700
EC00965=0.4023,1826.4284
EC00966=1.5064,1828.1658
EC00967=3.2134,1829.7669
EC00968=5.3325,1831.0323
EC00969=7.8395,1832.0364
EC00970=10.4506,1833.0299
EC00971=12.6950,1834.2655
EC00972=14.1862,1836.0719
EC00973=14.7367,1838.7215
EC00974=14.7681,1841.7023
EC00975=14.7639,1845.0000
EC00976=14.7681,1848.2977
EC00977=14.7367,1851.2785
EC00978=14.1862,1853.9281
EC00979=12.6950,1855.7345
EC00980=10.4506,1856.9701
EC00981=7.8395,1857.9636
EC00982=5.3325,1858.9677
EC00983=3.2134,1860.2331
EC00984=1.5064,1861.8342
EC00985=0.4023,1863.5716
EC00986=0.0692,1865.2300
EC00987=0.0075,1866.7569
EC00988=0.0074,1868.2435
EC00989=0.0671,1869.7700
EC00990=0.4022,1871.4284
EC00991=1.5081,1873.1658
EC00992=3.2124,1874.7673
EC00993=5.3324,1876.0322
EC00994=7.8426,1877.0367
EC00995=10.4501,1878.0300
EC00996=12.6975,1879.2653
EC00997=14.1865,1881.0716
EC00998=14.7351,1883.7217
EC00999=14.7688,1886.7026
EC01000=17.7591,1890.0000
EC01001=17.7704,1893.2854
EC01002=17.7316,1896.2621
EC01003=17.0680,1898.9150
EC01004=15.2200,1900.7121
EC01005=12.3697,1901.9342
EC01006=9.1378,1902.9128
EC01007=6.1937,1903.8997
EC01008=3.7259,1905.1448
EC01009=1.7218,1906.7421
EC01010=0.4366,1908.4921
EC01011=0.0798,1910.1777
EC01012=0.0074,1911.7387
EC01013=0.0075,1913.2613
EC01014=0.0768,1914.8225
EC01015=0.4356,1916.5076
EC01016=1.7236,1918.2578
EC01017=3.7272,1919.8549
EC01018=6.1941,1921.1001
EC01019=9.1389,1922.0874
EC01020=12.3647,1923.0661
EC01021=15.2206,1924.2883
EC01022=17.0686,1926.0850
EC01023=17.7331,1928.7375
EC01024=17.7700,1931.7146
EC01025=17.7616,1935.0000
EC01026=17.7700,1938.2854
EC01027=17.7331,1941.2625
EC01028=17.0686,1943.9150
EC01029=15.2206,1945.7117
EC01030=12.3647,1946.9339
EC01031=9.1389,1947.9126
EC01032=6.1941,1948.8999
EC01033=3.7272,1950.1451
EC01034=1.7236,1951.7422
EC01035=0.4356,1953.4924
EC01036=0.0768,1955.1775
EC01037=0.0075,1956.7387
EC01038=0.0074,1958.2613
EC01039=0.0798,1959.8223
EC01040=0.4366,1961.5079
EC01041=1.7218,1963.2579
EC01042=3.7259,1964.8552
EC01043=6.1937,1966.1003
EC01044=9.1378,1967.0872
EC01045=12.3697,1968.0658
EC01046=15.2200,1969.2879
EC01047=17.0680,1971.0850
EC01048=17.7316,1973.7379
EC01049=17.7704,1976.7146
EC01050=17.7591,1980.0000
EC01051=17.7704,1983.2854
EC01052=17.7316,1986.2621
EC01053=17.0680,1988.9150
EC01054=15.2200,1990.7121
EC01055=12.3697,1991.9342
EC01056=9.1378,1992.9128
EC01057=6.1937,1993.8997
EC01058=3.7259,1995.1448
EC01059=1.7218,1996.7421
EC01060=0.4366,1998.4921
EC01061=0.0798,2000.1777
EC01062=0.0074,2001.7387
EC01063=0.0075,2003.2613
EC01064=0.0768,2004.8225
EC01065=0.4356,2006.5076
EC01066=1.7236,2008.2578
EC01067=3.7272,2009.8549
EC01068=6.1941,2011.1001
EC01069=9.1389,2012.0874
EC01070=12.3647,2013.0661
EC01071=15.2206,2014.2883
EC01072=17.0686,2016.0850
EC01073=17.7331,2018.7375
EC01074=17.7700,2021.7146
EC01075=17.7616,2025.0000
EC01076=17.7700,2028.2854
EC01077=17.7331,2031.2625
EC01078=17.0686,2033.9150
EC01079=15.2206,2035.7117
EC01080=12.3647,2036.9339
EC01081=9.1389,2037.9126
EC01082=6.1941,2038.8999
EC01083=3.7272,2040.1451
EC01084=1.7236,2041.7422
EC01085=0.4356,2043.4924
EC01086=0.0768,2045.1775
EC01087=0.0075,2046.7387
EC01088=0.0074,2048.2613
EC01089=0.0798,2049.8223
EC01090=0.4366,2051.5079
EC01091=1.7218,2053.2579
EC01092=3.7259,2054.8552
EC01093=6.1937,2056.1003
EC01094=9.1378,2057.0872
EC01095=12.3697,2058.0658
EC01096=15.2200,2059.2879
EC01097=17.0680,2061.0850
EC01098=17.7316,2063.7379
EC01099=17.7704,2066.7146
EC01100=17.7591,2070.0000
EC01101=17.7704,2073.2854
EC01102=17.7316,2076.2621
EC01103=17.0680,2078.9150
EC01104=15.2200,2080.7121
EC01105=12.3697,2081.9342
EC01106=9.1378,2082.9128
EC01107=6.1937,2083.8997
EC01108=3.7259,2085.1448
EC01109=1.7218,2086.7421
EC01110=0.4366,2088.4921
EC01111=0.0798,2090.1777
EC01112=0.0074,2091.7387
EC01113=0.0075,2093.2613
EC01114=0.0768,2094.8225
EC01115=0.4356,2096.5076
EC01116=1.7236,2098.2578
EC01117=3.7272,2099.8549
EC01118=6.1941,2101.1001
EC01119=9.1389,2102.0874
EC01120=12.3647,2103.0661
EC01121=15.2206,2104.2883
EC01122=17.0686,2106.0850
EC01123=17.7331,2108.7375
EC01124=17.7700,2111.7146
EC01125=17.7616,2115.0000
EC01126=17.7700,2118.2854
EC01127=17.7331,2121.2625
EC01128=17.0686,2123.9150
EC01129=15.2206,2125.7117
EC01130=12.3647,2126.9339
EC01131=9.1389,2127.9126
EC01132=6.1941,2128.8999
EC01133=3.7272,2130.1451
EC01134=1.7236,2131.7422
EC01135=0.4356,2133.4924
EC01136=0.0768,2135.1775
EC01137=0.0075,2136.7387
EC01138=0.0074,2138.2613
EC01139=0.0798,2139.8223
EC01140=0.4366,2141.5079
EC01141=1.7218,2143.2579
EC01142=3.7259,2144.8552
EC01143=6.1937,2146.1003
EC01144=9.1378,2147.0872
EC01145=12.3697,2148.0658
EC01146=15.2200,2149.2879
EC01147=17.0680,2151.0850
EC01148=17.7316,2153.7379
EC01149=17.7704,2156.7146
EC01150=17.7591,2160.0000
EC01151=17.7704,2163.2854
EC01152=17.7316,2166.2621
EC01153=17.0680,2168.9150
EC01154=15.2200,2170.7121
EC01155=12.3697,2171.9342
EC01156=9.1378,2172.9128
EC01157=6.1937,2173.8997
EC01158=3.7259,2175.1448
EC01159=1.7218,2176.7421
EC01160=0.4366,2178.4921
EC01161=0.0798,2180.1777
EC01162=0.0074,2181.7387
EC01163=0.0075,2183.2613
EC01164=0.0768,2184.8225
EC01165=0.4356,2186.5076
EC01166=1.7236,2188.2578
EC01167=3.7272,2189.8549
EC01168=6.1941,2191.1001
EC01169=9.1389,2192.0874
EC01170=12.3647,2193.0661
EC01171=15.2206,2194.2883
EC01172=17.0686,2196.0850
EC01173=17.7331,2198.7375
EC01174=17.7700,2201.7146
EC01175=17.7616,2205.0000
EC01176=17.7700,2208.2854
EC01177=17.7331,2211.2625
EC01178=17.0686,2213.9150
EC01179=15.2206,2215.7117
EC01180=12.3647,2216.9339
EC01181=9.1389,2217.9126
EC01182=6.1941,2218.8999
EC01183=3.7272,2220.1451
EC01184=1.7236,2221.7422
EC01185=0.4356,2223.4924
EC01186=0.0768,2225.1775
EC01187=0.0075,2226.7387
EC01188=0.0074,2228.2613
EC01189=0.0798,2229.8223
EC01190=0.4366,2231.5079
EC01191=1.7218,2233.2579
EC01192=3.7259,2234.8552
EC01193=6.1937,2236.1003
EC01194=9.1378,2237.0872
EC01195=12.3697,2238.0658
EC01196=15.2200,2239.2879
EC01197=17.0680,2241.0850
EC01198=17.7316,2243.7379
EC01199=17.7704,2246.7146
EC01200=20.4756,2250.0000
EC01201=20.4854,2253.2709
EC01202=20.4405,2256.2435
EC01203=19.6670,2258.8988
EC01204=17.4078,2260.6850
EC01205=13.8489,2261.8912
EC01206=9.9912,2262.8520
EC01207=6.7582,2263.8189
EC01208=4.0853,2265.0400
EC01209=1.8598,2266.6318
EC01210=0.4457,2268.3974
EC01211=0.0798,2270.1155
EC01212=0.0128,2271.7171
EC01213=0.0128,2273.2826
EC01214=0.0820,2274.8847
EC01215=0.4459,2276.6022
EC01216=1.8589,2278.3677
EC01217=4.0858,2279.9600
EC01218=6.7570,2281.1815
EC01219=9.9939,2282.1481
EC01220=13.8526,2283.1089
EC01221=17.4102,2284.3149
EC01222=19.6676,2286.1008
EC01223=20.4407,2288.7567
EC01224=20.4843,2291.7290
EC01225=20.4721,2295.0000
EC01226=20.4843,2298.2710
EC01227=20.4407,2301.2433
EC01228=19.6676,2303.8992
EC01229=17.4102,2305.6851
EC01230=13.8526,2306.8911
EC01231=9.9939,2307.8519
EC01232=6.7570,2308.8185
EC01233=4.0858,2310.0400
EC01234=1.8589,2311.6323
EC01235=0.4459,2313.3978
EC01236=0.0820,2315.1153
EC01237=0.0128,2316.7174
EC01238=0.0128,2318.2829
EC01239=0.0798,2319.8845
EC01240=0.4457,2321.6026
EC01241=1.8598,2323.3682
EC01242=4.0853,2324.9600
EC01243=6.7582,2326.1811
EC01244=9.9912,2327.1480
EC01245=13.8489,2328.1088
EC01246=17.4078,2329.3150
EC01247=19.6670,2331.1012
EC01248=20.4405,2333.7565
EC01249=20.4854,2336.7291
EC01250=20.4756,2340.0000
EC01251=20.4854,2343.2709
EC01252=20.4405,2346.2435
EC01253=19.6670,2348.8988
EC01254=17.4078,2350.6850
EC01255=13.8489,2351.8912
EC01256=9.9912,2352.8520
EC01257=6.7582,2353.8189
EC01258=4.0853,2355.0400
EC01259=1.8598,2356.6318
EC01260=0.4457,2358.3974
EC01261=0.0798,2360.1155
EC01262=0.0128,2361.7171
EC01263=0.0128,2363.2826
EC01264=0.0820,2364.8847
EC01265=0.4459,2366.6022
EC01266=1.8589,2368.3677
EC01267=4.0858,2369.9600
EC01268=6.7570,2371.1815
EC01269=9.9939,2372.1481
EC01270=13.8526,2373.1089
EC01271=17.4102,2374.3149
EC01272=19.6676,2376.1008
EC01273=20.4407,2378.7567
EC01274=20.4843,2381.7290
EC01275=20.4721,2385.0000
EC01276=20.4843,2388.2710
EC01277=20.4407,2391.2433
EC01278=19.6676,2393.8992
EC01279=17.4102,2395.6851
EC01280=13.8526,2396.8911
EC01281=9.9939,2397.8519
EC01282=6.7570,2398.8185
EC01283=4.0858,2400.0400
EC01284=1.8589,2401.6323
EC01285=0.4459,2403.3978
EC01286=0.0820,2405.1153
EC01287=0.0128,2406.7174
EC01288=0.0128,2408.2829
EC01289=0.0798,2409.8845
EC01290=0.4457,2411.6026
EC01291=1.8598,2413.3682
EC01292=4.0853,2414.9600
EC01293=6.7582,2416.1811
EC01294=9.9912,2417.1480
EC01295=13.8489,2418.1088
EC01296=17.4078,2419.3150
EC01297=19.6670,2421.1012
EC01298=20.4405,2423.7565
EC01299=20.4854,2426.7291
EC01300=20.4756,2430.0000
EC01301=20.4854,2433.2709
EC01302=20.4405,2436.2435
EC01303=19.6670,2438.8988
EC01304=17.4078,2440.6850
EC01305=13.8489,2441.8912
EC01306=9.9912,2442.8520
EC01307=6.7582,2443.8189
EC01308=4.0853,2445.0400
EC01309=1.8598,2446.6318
EC01310=0.4457,2448.3974
EC01311=0.0798,2450.1155
EC01312=0.0128,2451.7171
EC01313=0.0128,2453.2826
EC01314=0.0820,2454.8847
EC01315=0.4459,2456.6022
EC01316=1.8589,2458.3677
EC01317=4.0858,2459.9600
EC01318=6.7570,2461.1815
EC01319=9.9939,2462.1481
EC01320=13.8526,2463.1089
EC01321=17.4102,2464.3149
EC01322=19.6676,2466.1008
EC01323=20.4407,2468.7567
EC01324=20.4843,2471.7290
EC01325=20.4721,2475.0000
EC01326=20.4843,2478.2710
EC01327=20.4407,2481.2433
EC01328=19.6676,2483.8992
EC01329=17.4102,2485.6851
EC01330=13.8526,2486.8911
EC01331=9.9939,2487.8519
EC01332=6.7570,2488.8185
EC01333=4.0858,2490.0400
EC01334=1.8589,2491.6323
EC01335=0.4459,2493.3978
EC01336=0.0820,2495.1153
EC01337=0.0128,2496.7174
EC01338=0.0128,2498.2829
EC01339=0.0798,2499.8845
EC01340=0.4457,2501.6026
EC01341=1.8598,2503.3682
EC01342=4.0853,2504.9600
EC01343=6.7582,2506.1811
EC01344=9.9912,2507.1480
EC01345=13.8489,2508.1088
EC01346=17.4078,2509.3150
EC01347=19.6670,2511.1012
EC01348=20.4405,2513.7565
EC01349=20.4854,2516.7291
EC01350=20.4756,2520.0000
EC01351=20.4854,2523.2709
EC01352=20.4405,2526.2435
EC01353=19.6670,2528.8988
EC01354=17.4078,2530.6850
EC01355=13.8489,2531.8912
EC01356=9.9912,2532.8520
EC01357=6.7582,2533.8189
EC01358=4.0853,2535.0400
EC01359=1.8598,2536.6318
EC01360=0.4457,2538.3974
EC01361=0.0798,2540.1155
EC01362=0.0128,2541.7171
EC01363=0.0128,2543.2826
EC01364=0.0820,2544.8847
EC01365=0.4459,2546.6022
EC01366=1.8589,2548.3677
EC01367=4.0858,2549.9600
EC01368=6.7570,2551.1815
EC01369=9.9939,2552.1481
EC01370=13.8526,2553.1089
EC01371=17.4102,2554.3149
EC01372=19.6676,2556.1008
EC01373=20.4407,2558.7567
EC01374=20.4843,2561.7290
EC01375=20.4721,2565.0000
EC01376=20.4843,2568.2710
EC01377=20.4407,2571.2433
EC01378=19.6676,2573.8992
EC01379=17.4102,2575.6851
EC01380=13.8526,2576.8911
EC01381=9.9939,2577.8519
EC01382=6.7570,2578.8185
EC01383=4.0858,2580.0400
EC01384=1.8589,2581.6323
EC01385=0.4459,2583.3978
EC01386=0.0820,2585.1153
EC01387=0.0128,2586.7174
EC01388=0.0128,2588.2829
EC01389=0.0798,2589.8845
EC01390=0.4457,2591.6026
EC01391=1.8598,2593.3682
EC01392=4.0853,2594.9600
EC01393=6.7582,2596.1811
EC01394=9.9912,2597.1480
EC01395=13.8489,2598.1088
EC01396=17.4078,2599.3150
EC01397=19.6670,2601.1012
EC01398=20.4405,2603.7565
EC01399=20.4854,2606.7291
EC01400=22.9187,2610.0000
EC01401=22.9316,2613.2546
EC01402=22.8765,2616.2211
EC01403=21.9924,2618.8807
EC01404=19.2373,2620.6541
EC01405=14.8082,2621.8420
EC01406=10.3073,2622.7823
EC01407=6.9686,2623.7251
EC01408=4.2642,2624.9190
EC01409=1.9061,2626.5054
EC01410=0.4204,2628.2889
EC01411=0.0852,2630.0438
EC01412=0.0128,2631.6927
EC01413=0.0128,2633.3075
EC01414=0.0820,2634.9564
EC01415=0.4177,2636.7113
EC01416=1.9077,2638.4943
EC01417=4.2648,2640.0807
EC01418=6.9647,2641.2747
EC01419=10.3085,2642.2172
EC01420=14.8105,2643.1579
EC01421=19.2366,2644.3457
EC01422=21.9938,2646.1194
EC01423=22.8755,2648.7787
EC01424=22.9306,2651.7455
EC01425=22.9226,2655.0000
EC01426=22.9306,2658.2545
EC01427=22.8755,2661.2213
EC01428=21.9938,2663.8806
EC01429=19.2366,2665.6543
EC01430=14.8105,2666.8421
EC01431=10.3085,2667.7828
EC01432=6.9647,2668.7253
EC01433=4.2648,2669.9193
EC01434=1.9077,2671.5057
EC01435=0.4177,2673.2887
EC01436=0.0820,2675.0436
EC01437=0.0128,2676.6925
EC01438=0.0128,2678.3073
EC01439=0.0852,2679.9562
EC01440=0.4204,2681.7111
EC01441=1.9061,2683.4946
EC01442=4.2642,2685.0810
EC01443=6.9686,2686.2749
EC01444=10.3073,2687.2177
EC01445=14.8082,2688.1580
EC01446=19.2373,2689.3459
EC01447=21.9924,2691.1193
EC01448=22.8765,2693.7789
EC01449=22.9316,2696.7454
EC01450=22.9187,2700.0000
EC01451=22.9316,2703.2546
EC01452=22.8765,2706.2211
EC01453=21.9924,2708.8807
EC01454=19.2373,2710.6541
EC01455=14.8082,2711.8420
EC01456=10.3073,2712.7823
EC01457=6.9686,2713.7251
EC01458=4.2642,2714.9190
EC01459=1.9061,2716.5054
EC01460=0.4204,2718.2889
EC01461=0.0852,2720.0438
EC01462=0.0128,2721.6927
EC01463=0.0128,2723.3075
EC01464=0.0820,2724.9564
EC01465=0.4177,2726.7113
EC01466=1.9077,2728.4943
EC01467=4.2648,2730.0807
EC01468=6.9647,2731.2747
EC01469=10.3085,2732.2172
EC01470=14.8105,2733.1579
EC01471=19.2366,2734.3457
EC01472=21.9938,2736.1194
EC01473=22.8755,2738.7787
EC01474=22.9306,2741.7455
EC01475=22.9226,2745.0000
EC01476=22.9306,2748.2545
EC01477=22.8755,2751.2213
EC01478=21.9938,2753.8806
EC01479=19.2366,2755.6543
EC01480=14.8105,2756.8421
EC01481=10.3085,2757.7828
EC01482=6.9647,2758.7253
EC01483=4.2648,2759.9193
EC01484=1.9077,2761.5057
EC01485=0.4177,2763.2887
EC01486=0.0820,2765.0436
EC01487=0.0128,2766.6925
EC01488=0.0128,2768.3073
EC01489=0.0852,2769.9562
EC01490=0.4204,2771.7111
EC01491=1.9061,2773.4946
EC01492=4.2642,2775.0810
EC01493=6.9686,2776.2749
EC01494=10.3073,2777.2177
EC01495=14.8082,2778.1580
EC01496=19.2373,2779.3459
EC01497=21.9924,2781.1193
EC01498=22.8765,2783.7789
EC01499=22.9316,2786.7454
EC01500=22.9187,2790.0000
EC01501=22.9316,2793.2546
EC01502=22.8765,2796.2211
EC01503=21.9924,2798.8807
EC01504=19.2373,2800.6541
EC01505=14.8082,2801.8420
EC01506=10.3073,2802.7823
EC01507=6.9686,2803.7251
EC01508=4.2642,2804.9190
EC01509=1.9061,2806.5054
EC01510=0.4204,2808.2889
EC01511=0.0852,2810.0438
EC01512=0.0128,2811.6927
EC01513=0.0128,2813.3075
EC01514=0.0820,2814.9564
EC01515=0.4177,2816.7113
EC01516=1.9077,2818.4943
EC01517=4.2648,2820.0807
EC01518=6.9647,2821.2747
EC01519=10.3085,2822.2172
EC01520=14.8105,2823.1579
EC01521=19.2366,2824.3457
EC01522=21.9938,2826.1194
EC01523=22.8755,2828.7787
EC01524=22.9306,2831.7455
EC01525=22.9226,2835.0000
EC01526=22.9306,2838.2545
EC01527=22.8755,2841.2213
EC01528=21.9938,2843.8806
EC01529=19.2366,2845.6543
EC01530=14.8105,2846.8421
EC01531=10.3085,2847.7828
EC01532=6.9647,2848.7253
EC01533=4.2648,2849.9193
EC01534=1.9077,2851.5057
EC01535=0.4177,2853.2887
EC01536=0.0820,2855.0436
EC01537=0.0128,2856.6925
EC01538=0.0128,2858.3073
EC01539=0.0852,2859.9562
EC01540=0.4204,2861.7111
EC01541=1.9061,2863.4946
EC01542=4.2642,2865.0810
EC01543=6.9686,2866.2749
EC01544=10.3073,2867.2177
EC01545=14.8082,2868.1580
EC01546=19.2373,2869.3459
EC01547=21.9924,2871.1193
EC01548=22.8765,2873.7789
EC01549=22.9316,2876.7454
EC01550=22.9187,2880.0000
EC01551=22.9316,2883.2546
EC01552=22.8765,2886.2211
EC01553=21.9924,2888.8807
EC01554=19.2373,2890.6541
EC01555=14.8082,2891.8420
EC01556=10.3073,2892.7823
EC01557=6.9686,2893.7251
EC01558=4.2642,2894.9190
EC01559=1.9061,2896.5054
EC01560=0.4204,2898.2889
EC01561=0.0852,2900.0438
EC01562=0.0128,2901.6927
EC01563=0.0128,2903.3075
EC01564=0.0820,2904.9564
EC01565=0.4177,2906.7113
EC01566=1.9077,2908.4943
EC01567=4.2648,2910.0807
EC01568=6.9647,2911.2747
EC01569=10.3085,2912.2172
EC01570=14.8105,2913.1579
EC01571=19.2366,2914.3457
EC01572=21.9938,2916.1194
EC01573=22.8755,2918.7787
EC01574=22.9306,2921.7455
EC01575=22.9226,2925.0000
EC01576=22.9306,2928.2545
EC01577=22.8755,2931.2213
EC01578=21.9938,2933.8806
EC01579=19.2366,2935.6543
EC01580=14.8105,2936.8421
EC01581=10.3085,2937.7828
EC01582=6.9647,2938.7253
EC01583=4.2648,2939.9193
EC01584=1.9077,2941.5057
EC01585=0.4177,2943.2887
EC01586=0.0820,2945.0436
EC01587=0.0128,2946.6925
EC01588=0.0128,2948.3073
EC01589=0.0852,2949.9562
EC01590=0.4204,2951.7111
EC01591=1.9061,2953.4946
EC01592=4.2642,2955.0810
EC01593=6.9686,2956.2749
EC01594=10.3073,2957.2177
EC01595=14.8082,2958.1580
EC01596=19.2373,2959.3459
EC01597=21.9924,2961.1193
EC01598=22.8765,2963.7789
EC01599=22.9316,2966.7454
EC01600=25.1121,2970.0000
EC01601=25.1250,2973.2359
EC01602=25.0665,2976.1970
EC01603=24.0583,2978.8601
EC01604=20.6589,2980.6197
EC01605=15.1715,2981.7864
EC01606=10.0480,2982.7041
EC01607=6.7819,2983.6200
EC01608=4.2461,2984.7831
EC01609=1.8706,2986.3632
EC01610=0.3589,2988.1666
EC01611=0.0798,2989.9634
EC01612=0.0074,2991.6649
EC01613=0.0075,2993.3352
EC01614=0.0820,2995.0366
EC01615=0.3614,2996.8332
EC01616=1.8693,2998.6370
EC01617=4.2497,3000.2167
EC01618=6.7838,3001.3801
EC01619=10.0525,3002.2959
EC01620=15.1731,3003.2134
EC01621=20.6601,3004.3801
EC01622=24.0591,3006.1402
EC01623=25.0675,3008.8032
EC01624=25.1255,3011.7642
EC01625=25.1124,3015.0000
EC01626=25.1255,3018.2358
EC01627=25.0675,3021.1968
EC01628=24.0591,3023.8598
EC01629=20.6601,3025.6199
EC01630=15.1731,3026.7866
EC01631=10.0525,3027.7041
EC01632=6.7838,3028.6199
EC01633=4.2497,3029.7833
EC01634=1.8693,3031.3630
EC01635=0.3614,3033.1668
EC01636=0.0820,3034.9634
EC01637=0.0075,3036.6648
EC01638=0.0074,3038.3351
EC01639=0.0798,3040.0366
EC01640=0.3589,3041.8334
EC01641=1.8706,3043.6368
EC01642=4.2461,3045.2169
EC01643=6.7819,3046.3800
EC01644=10.0480,3047.2959
EC01645=15.1715,3048.2136
EC01646=20.6589,3049.3803
EC01647=24.0583,3051.1399
EC01648=25.0665,3053.8030
EC01649=25.1250,3056.7641
EC01650=25.1121,3060.0000
EC01651=25.1250,3063.2359
EC01652=25.0665,3066.1970
EC01653=24.0591,3068.8601
EC01654=20.6589,3070.6197
EC01655=15.1715,3071.7864
EC01656=10.0480,3072.7041
EC01657=6.7819,3073.6200
EC01658=4.2461,3074.7831
EC01659=1.8706,3076.3632
EC01660=0.3589,3078.1666
EC01661=0.0798,3079.9634
EC01662=0.0074,3081.6649
EC01663=0.0075,3083.3352
EC01664=0.0820,3085.0366
EC01665=0.3614,3086.8332
EC01666=1.8693,3088.6370
EC01667=4.2497,3090.2167
EC01668=6.7838,3091.3801
EC01669=10.0525,3092.2959
EC01670=15.1731,3093.2134
EC01671=20.6601,3094.3801
EC01672=24.0591,3096.1402
EC01673=25.0675,3098.8032
EC01674=25.1255,3101.7642
EC01675=25.1124,3105.0000
EC01676=25.1255,3108.2358
EC01677=25.0675,3111.1968
EC01678=24.0591,3113.8598
EC01679=20.6601,3115.6199
EC01680=15.1731,3116.7866
EC01681=10.0525,3117.7041
EC01682=6.7838,3118.6199
EC01683=4.2497,3119.7833
EC01684=1.8693,3121.3630
EC01685=0.3614,3123.1668
EC01686=0.0820,3124.9634
EC01687=0.0075,3126.6648
EC01688=0.0074,3128.3351
EC01689=0.0798,3130.0366
EC01690=0.3589,3131.8334
EC01691=1.8706,3133.6368
EC01692=4.2461,3135.2169
EC01693=6.7819,3136.3800
EC01694=10.0480,3137.2959
EC01695=15.1715,3138.2136
EC01696=20.6589,3139.3803
EC01697=24.0583,3141.1399
EC01698=25.0665,3143.8030
EC01699=25.1250,3146.7641
EC01700=25.1121,3150.0000
EC01701=25.1250,3153.2359
EC01702=25.0665,3156.1970
EC01703=24.0591,3158.8601
EC01704=20.6589,3160.6197
EC01705=15.1715,3161.7864
EC01706=10.0480,3162.7041
EC01707=6.7819,3163.6200
EC01708=4.2461,3164.7831
EC01709=1.8706,3166.3632
EC01710=0.3589,3168.1666
EC01711=0.0798,3169.9634
EC01712=0.0074,3171.6649
EC01713=0.0075,3173.3352
EC01714=0.0820,3175.0366
EC01715=0.3614,3176.8332
EC01716=1.8693,3178.6370
EC01717=4.2497,3180.2167
EC01718=6.7838,3181.3801
EC01719=10.0525,3182.2959
EC01720=15.1731,3183.2134
EC01721=20.6601,3184.3801
EC01722=24.0591,3186.1402
EC01723=25.0675,3188.8032
EC01724=25.1255,3191.7642
EC01725=25.1124,3195.0000
EC01726=25.1255,3198.2358
EC01727=25.0675,3201.1968
EC01728=24.0591,3203.8598
EC01729=20.6601,3205.6199
EC01730=15.1731,3206.7866
EC01731=10.0525,3207.7041
EC01732=6.7838,3208.6199
EC01733=4.2497,3209.7833
EC01734=1.8693,3211.3630
EC01735=0.3614,3213.1668
EC01736=0.0820,3214.9634
EC01737=0.0075,3216.6648
EC01738=0.0074,3218.3351
EC01739=0.0798,3220.0366
EC01740=0.3589,3221.8334
EC01741=1.8706,3223.6368
EC01742=4.2461,3225.2169
EC01743=6.7819,3226.3800
EC01744=10.0480,3227.2959
EC01745=15.1715,3228.2136
EC01746=20.6589,3229.3803
EC01747=24.0583,3231.1399
EC01748=25.0665,3233.8030
EC01749=25.1250,3236.7641
EC01750=25.1121,3240.0000
EC01751=25.1250,3243.2359
EC01752=25.0665,3246.1970
EC01753=24.0591,3248.8601
EC01754=20.6589,3250.6197
EC01755=15.1715,3251.7864
EC01756=10.0480,3252.7041
EC01757=6.7819,3253.6200
EC01758=4.2461,3254.7831
EC01759=1.8706,3256.3632
EC01760=0.3589,3258.1666
EC01761=0.0798,3259.9634
EC01762=0.0074,3261.6649
EC01763=0.0075,3263.3352
EC01764=0.0820,3265.0366
EC01765=0.3614,3266.8332
EC01766=1.8693,3268.6370
EC01767=4.2497,3270.2167
EC01768=6.7838,3271.3801
EC01769=10.0525,3272.2959
EC01770=15.1731,3273.2134
EC01771=20.6601,3274.3801
EC01772=24.0591,3276.1402
EC01773=25.0675,3278.8032
EC01774=25.1255,3281.7642
EC01775=25.1124,3285.0000
EC01776=25.1255,3288.2358
EC01777=25.0675,3291.1968
EC01778=24.0591,3293.8598
EC01779=20.6601,3295.6199
EC01780=15.1731,3296.7866
EC01781=10.0525,3297.7041
EC01782=6.7838,3298.6199
EC01783=4.2497,3299.7833
EC01784=1.8693,3301.3630
EC01785=0.3614,3303.1668
EC01786=0.0820,3304.9634
EC01787=0.0075,3306.6648
EC01788=0.0074,3308.3351
EC01789=0.0798,3310.0366
EC01790=0.3589,3311.8334
EC01791=1.8706,3313.6368
EC01792=4.2461,3315.2169
EC01793=6.7819,3316.3800
EC01794=10.0480,3317.2959
EC01795=15.1715,3318.2136
EC01796=20.6589,3319.3803
EC01797=24.0591,3321.1399
EC01798=25.0665,3323.8030
EC01799=25.1250,3326.7641
EC01800=27.0775,3330.0000
EC01801=27.0874,3333.2152
EC01802=27.0185,3336.1699
EC01803=25.8724,3338.8371
EC01804=21.6484,3340.5819
EC01805=14.9094,3341.7253
EC01806=9.2462,3342.6169
EC01807=6.2189,3343.5035
EC01808=4.0294,3344.6333
EC01809=1.7445,3346.2063
EC01810=0.2756,3348.0324
EC01811=0.0778,3349.8748
EC01812=0.0074,3351.6343
EC01813=0.0075,3353.3660
EC01814=0.0768,3355.1253
EC01815=0.2718,3356.9678
EC01816=1.7463,3358.7935
EC01817=4.0258,3360.3670
EC01818=6.2165,3361.4965
EC01819=9.2440,3362.3830
EC01820=14.9062,3363.2751
EC01821=21.6521,3364.4183
EC01822=25.8712,3366.1625
EC01823=27.0203,3368.8301
EC01824=27.0876,3371.7846
EC01825=27.0793,3375.0000
EC01826=27.0876,3378.2154
EC01827=27.0203,3381.1699
EC01828=25.8712,3383.8375
EC01829=21.6521,3385.5817
EC01830=14.9062,3386.7249
EC01831=9.2440,3387.6170
EC01832=6.2165,3388.5035
EC01833=4.0258,3389.6330
EC01834=1.7463,3391.2065
EC01835=0.2718,3393.0322
EC01836=0.0768,3394.8747
EC01837=0.0075,3396.6340
EC01838=0.0074,3398.3657
EC01839=0.0778,3400.1252
EC01840=0.2756,3401.9676
EC01841=1.7445,3403.7937
EC01842=4.0294,3405.3667
EC01843=6.2189,3406.4965
EC01844=9.2462,3407.3831
EC01845=14.9094,3408.2747
EC01846=21.6484,3409.4181
EC01847=25.8724,3411.1629
EC01848=27.0185,3413.8301
EC01849=27.0874,3416.7848
EC01850=27.0775,3420.0000
EC01851=27.0874,3423.2152
EC01852=27.0185,3426.1699
EC01853=25.8724,3428.8371
EC01854=21.6484,3430.5819
EC01855=14.9094,3431.7253
EC01856=9.2462,3432.6169
EC01857=6.2189,3433.5035
EC01858=4.0294,3434.6333
EC01859=1.7445,3436.2063
EC01860=0.2756,3438.0324
EC01861=0.0778,3439.8748
EC01862=0.0074,3441.6343
EC01863=0.0075,3443.3660
EC01864=0.0768,3445.1253
EC01865=0.2718,3446.9678
EC01866=1.7463,3448.7935
EC01867=4.0258,3450.3670
EC01868=6.2165,3451.4965
EC01869=9.2440,3452.3830
EC01870=14.9062,3453.2751
EC01871=21.6521,3454.4183
EC01872=25.8712,3456.1625
EC01873=27.0203,3458.8301
EC01874=27.0876,3461.7846
EC01875=27.0793,3465.0000
EC01876=27.0876,3468.2154
EC01877=27.0203,3471.1699
EC01878=25.8712,3473.8375
EC01879=21.6521,3475.5817
EC01880=14.9062,3476.7249
EC01881=9.2440,3477.6170
EC01882=6.2165,3478.5035
EC01883=4.0258,3479.6330
EC01884=1.7463,3481.2065
EC01885=0.2718,3483.0322
EC01886=0.0768,3484.8747
EC01887=0.0075,3486.6340
EC01888=0.0074,3488.3657
EC01889=0.0778,3490.1252
EC01890=0.2756,3491.9676
EC01891=1.7445,3493.7937
EC01892=4.0294,3495.3667
EC01893=6.2189,3496.4965
EC01894=9.2462,3497.3831
EC01895=14.9094,3498.2747
EC01896=21.6484,3499.4181
EC01897=25.8724,3501.1629
EC01898=27.0185,3503.8301
EC01899=27.0874,3506.7848
EC01900=27.0775,3510.0000
EC01901=27.0874,3513.2152
EC01902=27.0185,3516.1699
EC01903=25.8724,3518.8371
EC01904=21.6484,3520.5819
EC01905=14.9094,3521.7253
EC01906=9.2462,3522.6169
EC01907=6.2189,3523.5035
EC01908=4.0294,3524.6333
EC01909=1.7445,3526.2063
EC01910=0.2756,3528.0324
EC01911=0.0778,3529.8748
EC01912=0.0074,3531.6343
EC01913=0.0075,3533.3660
EC01914=0.0768,3535.1253
EC01915=0.2718,3536.9678
EC01916=1.7463,3538.7935
EC01917=4.0258,3540.3670
EC01918=6.2165,3541.4965
EC01919=9.2440,3542.3830
EC01920=14.9062,3543.2751
EC01921=21.6521,3544.4183
EC01922=25.8712,3546.1625
EC01923=27.0203,3548.8301
EC01924=27.0876,3551.7846
EC01925=27.0793,3555.0000
EC01926=27.0876,3558.2154
EC01927=27.0203,3561.1699
EC01928=25.8712,3563.8375
EC01929=21.6521,3565.5817
EC01930=14.9062,3566.7249
EC01931=9.2440,3567.6170
EC01932=6.2165,3568.5035
EC01933=4.0258,3569.6330
EC01934=1.7463,3571.2065
EC01935=0.2718,3573.0322
EC01936=0.0768,3574.8747
EC01937=0.0075,3576.6340
EC01938=0.0074,3578.3657
EC01939=0.0778,3580.1252
EC01940=0.2756,3581.9676
EC01941=1.7445,3583.7937
EC01942=4.0294,3585.3667
EC01943=6.2189,3586.4965
EC01944=9.2462,3587.3831
EC01945=14.9094,3588.2747
EC01946=21.6484,3589.4181
EC01947=25.8724,3591.1629
EC01948=27.0185,3593.8301
EC01949=27.0874,3596.7848
EC01950=27.0775,3600.0000
EC01951=27.0874,3603.2152
EC01952=27.0185,3606.1699
EC01953=25.8724,3608.8371
EC01954=21.6484,3610.5819
EC01955=14.9094,3611.7253
EC01956=9.2462,3612.6169
EC01957=6.2189,3613.5035
EC01958=4.0294,3614.6333
EC01959=1.7445,3616.2063
EC01960=0.2756,3618.0324
EC01961=0.0778,3619.8748
EC01962=0.0074,3621.6343
EC01963=0.0075,3623.3660
EC01964=0.0768,3625.1253
EC01965=0.2718,3626.9678
EC01966=1.7463,3628.7935
EC01967=4.0258,3630.3670
EC01968=6.2165,3631.4965
EC01969=9.2440,3632.3830
EC01970=14.9062,3633.2751
EC01971=21.6521,3634.4183
EC01972=25.8712,3636.1625
EC01973=27.0203,3638.8301
EC01974=27.0876,3641.7846
EC01975=27.0793,3645.0000
EC01976=27.0876,3648.2154
EC01977=27.0203,3651.1699
EC01978=25.8712,3653.8375
EC01979=21.6521,3655.5817
EC01980=14.9062,3656.7249
EC01981=9.2440,3657.6170
EC01982=6.2165,3658.5035
EC01983=4.0258,3659.6330
EC01984=1.7463,3661.2065
EC01985=0.2718,3663.0322
EC01986=0.0768,3664.8747
EC01987=0.0075,3666.6340
EC01988=0.0074,3668.3657
EC01989=0.0778,3670.1252
EC01990=0.2756,3671.9676
EC01991=1.7445,3673.7937
EC01992=4.0294,3675.3667
EC01993=6.2189,3676.4965
EC01994=9.2462,3677.3831
EC01995=14.9094,3678.2747
EC01996=21.6484,3679.4181
EC01997=25.8724,3681.1629
EC01998=27.0185,3683.8301
EC01999=27.0874,3686.7848
//INST
///DATE 2021/09/24 16:41
///COMM
///ATTR SC,RW,RJ
////FRAME USER 2
///GROUP1 RB1
///GROUP2 ST1
NOP
SMOVL C00000 +MOVJ EC00000
SPEED V=10.0
ARCON
SMOVL C00001 +MOVJ EC00001
SMOVL C00002 +MOVJ EC00002
SMOVL C00003 +MOVJ EC00003
SMOVL C00004 +MOVJ EC00004
SMOVL C00005 +MOVJ EC00005
SMOVL C00006 +MOVJ EC00006
SMOVL C00007 +MOVJ EC00007
SMOVL C00008 +MOVJ EC00008
SMOVL C00009 +MOVJ EC00009
SMOVL C00010 +MOVJ EC00010
SMOVL C00011 +MOVJ EC00011
SMOVL C00012 +MOVJ EC00012
SMOVL C00013 +MOVJ EC00013
SMOVL C00014 +MOVJ EC00014
SMOVL C00015 +MOVJ EC00015
SMOVL C00016 +MOVJ EC00016
SMOVL C00017 +MOVJ EC00017
SMOVL C00018 +MOVJ EC00018
SMOVL C00019 +MOVJ EC00019
SMOVL C00020 +MOVJ EC00020
SMOVL C00021 +MOVJ EC00021
SMOVL C00022 +MOVJ EC00022
SMOVL C00023 +MOVJ EC00023
SMOVL C00024 +MOVJ EC00024
SMOVL C00025 +MOVJ EC00025
SMOVL C00026 +MOVJ EC00026
SMOVL C00027 +MOVJ EC00027
SMOVL C00028 +MOVJ EC00028
SMOVL C00029 +MOVJ EC00029
SMOVL C00030 +MOVJ EC00030
SMOVL C00031 +MOVJ EC00031
SMOVL C00032 +MOVJ EC00032
SMOVL C00033 +MOVJ EC00033
SMOVL C00034 +MOVJ EC00034
SMOVL C00035 +MOVJ EC00035
SMOVL C00036 +MOVJ EC00036
SMOVL C00037 +MOVJ EC00037
SMOVL C00038 +MOVJ EC00038
SMOVL C00039 +MOVJ EC00039
SMOVL C00040 +MOVJ EC00040
SMOVL C00041 +MOVJ EC00041
SMOVL C00042 +MOVJ EC00042
SMOVL C00043 +MOVJ EC00043
SMOVL C00044 +MOVJ EC00044
SMOVL C00045 +MOVJ EC00045
SMOVL C00046 +MOVJ EC00046
SMOVL C00047 +MOVJ EC00047
SMOVL C00048 +MOVJ EC00048
SMOVL C00049 +MOVJ EC00049
SMOVL C00050 +MOVJ EC00050
SMOVL C00051 +MOVJ EC00051
SMOVL C00052 +MOVJ EC00052
SMOVL C00053 +MOVJ EC00053
SMOVL C00054 +MOVJ EC00054
SMOVL C00055 +MOVJ EC00055
SMOVL C00056 +MOVJ EC00056
SMOVL C00057 +MOVJ EC00057
SMOVL C00058 +MOVJ EC00058
SMOVL C00059 +MOVJ EC00059
SMOVL C00060 +MOVJ EC00060
SMOVL C00061 +MOVJ EC00061
SMOVL C00062 +MOVJ EC00062
SMOVL C00063 +MOVJ EC00063
SMOVL C00064 +MOVJ EC00064
SMOVL C00065 +MOVJ EC00065
SMOVL C00066 +MOVJ EC00066
SMOVL C00067 +MOVJ EC00067
SMOVL C00068 +MOVJ EC00068
SMOVL C00069 +MOVJ EC00069
SMOVL C00070 +MOVJ EC00070
SMOVL C00071 +MOVJ EC00071
SMOVL C00072 +MOVJ EC00072
SMOVL C00073 +MOVJ EC00073
SMOVL C00074 +MOVJ EC00074
SMOVL C00075 +MOVJ EC00075
SMOVL C00076 +MOVJ EC00076
SMOVL C00077 +MOVJ EC00077
SMOVL C00078 +MOVJ EC00078
SMOVL C00079 +MOVJ EC00079
SMOVL C00080 +MOVJ EC00080
SMOVL C00081 +MOVJ EC00081
SMOVL C00082 +MOVJ EC00082
SMOVL C00083 +MOVJ EC00083
SMOVL C00084 +MOVJ EC00084
SMOVL C00085 +MOVJ EC00085
SMOVL C00086 +MOVJ EC00086
SMOVL C00087 +MOVJ EC00087
SMOVL C00088 +MOVJ EC00088
SMOVL C00089 +MOVJ EC00089
SMOVL C00090 +MOVJ EC00090
SMOVL C00091 +MOVJ EC00091
SMOVL C00092 +MOVJ EC00092
SMOVL C00093 +MOVJ EC00093
SMOVL C00094 +MOVJ EC00094
SMOVL C00095 +MOVJ EC00095
SMOVL C00096 +MOVJ EC00096
SMOVL C00097 +MOVJ EC00097
SMOVL C00098 +MOVJ EC00098
SMOVL C00099 +MOVJ EC00099
SMOVL C00100 +MOVJ EC00100
SMOVL C00101 +MOVJ EC00101
SMOVL C00102 +MOVJ EC00102
SMOVL C00103 +MOVJ EC00103
SMOVL C00104 +MOVJ EC00104
SMOVL C00105 +MOVJ EC00105
SMOVL C00106 +MOVJ EC00106
SMOVL C00107 +MOVJ EC00107
SMOVL C00108 +MOVJ EC00108
SMOVL C00109 +MOVJ EC00109
SMOVL C00110 +MOVJ EC00110
SMOVL C00111 +MOVJ EC00111
SMOVL C00112 +MOVJ EC00112
SMOVL C00113 +MOVJ EC00113
SMOVL C00114 +MOVJ EC00114
SMOVL C00115 +MOVJ EC00115
SMOVL C00116 +MOVJ EC00116
SMOVL C00117 +MOVJ EC00117
SMOVL C00118 +MOVJ EC00118
SMOVL C00119 +MOVJ EC00119
SMOVL C00120 +MOVJ EC00120
SMOVL C00121 +MOVJ EC00121
SMOVL C00122 +MOVJ EC00122
SMOVL C00123 +MOVJ EC00123
SMOVL C00124 +MOVJ EC00124
SMOVL C00125 +MOVJ EC00125
SMOVL C00126 +MOVJ EC00126
SMOVL C00127 +MOVJ EC00127
SMOVL C00128 +MOVJ EC00128
SMOVL C00129 +MOVJ EC00129
SMOVL C00130 +MOVJ EC00130
SMOVL C00131 +MOVJ EC00131
SMOVL C00132 +MOVJ EC00132
SMOVL C00133 +MOVJ EC00133
SMOVL C00134 +MOVJ EC00134
SMOVL C00135 +MOVJ EC00135
SMOVL C00136 +MOVJ EC00136
SMOVL C00137 +MOVJ EC00137
SMOVL C00138 +MOVJ EC00138
SMOVL C00139 +MOVJ EC00139
SMOVL C00140 +MOVJ EC00140
SMOVL C00141 +MOVJ EC00141
SMOVL C00142 +MOVJ EC00142
SMOVL C00143 +MOVJ EC00143
SMOVL C00144 +MOVJ EC00144
SMOVL C00145 +MOVJ EC00145
SMOVL C00146 +MOVJ EC00146
SMOVL C00147 +MOVJ EC00147
SMOVL C00148 +MOVJ EC00148
SMOVL C00149 +MOVJ EC00149
SMOVL C00150 +MOVJ EC00150
SMOVL C00151 +MOVJ EC00151
SMOVL C00152 +MOVJ EC00152
SMOVL C00153 +MOVJ EC00153
SMOVL C00154 +MOVJ EC00154
SMOVL C00155 +MOVJ EC00155
SMOVL C00156 +MOVJ EC00156
SMOVL C00157 +MOVJ EC00157
SMOVL C00158 +MOVJ EC00158
SMOVL C00159 +MOVJ EC00159
SMOVL C00160 +MOVJ EC00160
SMOVL C00161 +MOVJ EC00161
SMOVL C00162 +MOVJ EC00162
SMOVL C00163 +MOVJ EC00163
SMOVL C00164 +MOVJ EC00164
SMOVL C00165 +MOVJ EC00165
SMOVL C00166 +MOVJ EC00166
SMOVL C00167 +MOVJ EC00167
SMOVL C00168 +MOVJ EC00168
SMOVL C00169 +MOVJ EC00169
SMOVL C00170 +MOVJ EC00170
SMOVL C00171 +MOVJ EC00171
SMOVL C00172 +MOVJ EC00172
SMOVL C00173 +MOVJ EC00173
SMOVL C00174 +MOVJ EC00174
SMOVL C00175 +MOVJ EC00175
SMOVL C00176 +MOVJ EC00176
SMOVL C00177 +MOVJ EC00177
SMOVL C00178 +MOVJ EC00178
SMOVL C00179 +MOVJ EC00179
SMOVL C00180 +MOVJ EC00180
SMOVL C00181 +MOVJ EC00181
SMOVL C00182 +MOVJ EC00182
SMOVL C00183 +MOVJ EC00183
SMOVL C00184 +MOVJ EC00184
SMOVL C00185 +MOVJ EC00185
SMOVL C00186 +MOVJ EC00186
SMOVL C00187 +MOVJ EC00187
SMOVL C00188 +MOVJ EC00188
SMOVL C00189 +MOVJ EC00189
SMOVL C00190 +MOVJ EC00190
SMOVL C00191 +MOVJ EC00191
SMOVL C00192 +MOVJ EC00192
SMOVL C00193 +MOVJ EC00193
SMOVL C00194 +MOVJ EC00194
SMOVL C00195 +MOVJ EC00195
SMOVL C00196 +MOVJ EC00196
SMOVL C00197 +MOVJ EC00197
SMOVL C00198 +MOVJ EC00198
SMOVL C00199 +MOVJ EC00199
SMOVL C00200 +MOVJ EC00200
SMOVL C00201 +MOVJ EC00201
SMOVL C00202 +MOVJ EC00202
SMOVL C00203 +MOVJ EC00203
SMOVL C00204 +MOVJ EC00204
SMOVL C00205 +MOVJ EC00205
SMOVL C00206 +MOVJ EC00206
SMOVL C00207 +MOVJ EC00207
SMOVL C00208 +MOVJ EC00208
SMOVL C00209 +MOVJ EC00209
SMOVL C00210 +MOVJ EC00210
SMOVL C00211 +MOVJ EC00211
SMOVL C00212 +MOVJ EC00212
SMOVL C00213 +MOVJ EC00213
SMOVL C00214 +MOVJ EC00214
SMOVL C00215 +MOVJ EC00215
SMOVL C00216 +MOVJ EC00216
SMOVL C00217 +MOVJ EC00217
SMOVL C00218 +MOVJ EC00218
SMOVL C00219 +MOVJ EC00219
SMOVL C00220 +MOVJ EC00220
SMOVL C00221 +MOVJ EC00221
SMOVL C00222 +MOVJ EC00222
SMOVL C00223 +MOVJ EC00223
SMOVL C00224 +MOVJ EC00224
SMOVL C00225 +MOVJ EC00225
SMOVL C00226 +MOVJ EC00226
SMOVL C00227 +MOVJ EC00227
SMOVL C00228 +MOVJ EC00228
SMOVL C00229 +MOVJ EC00229
SMOVL C00230 +MOVJ EC00230
SMOVL C00231 +MOVJ EC00231
SMOVL C00232 +MOVJ EC00232
SMOVL C00233 +MOVJ EC00233
SMOVL C00234 +MOVJ EC00234
SMOVL C00235 +MOVJ EC00235
SMOVL C00236 +MOVJ EC00236
SMOVL C00237 +MOVJ EC00237
SMOVL C00238 +MOVJ EC00238
SMOVL C00239 +MOVJ EC00239
SMOVL C00240 +MOVJ EC00240
SMOVL C00241 +MOVJ EC00241
SMOVL C00242 +MOVJ EC00242
SMOVL C00243 +MOVJ EC00243
SMOVL C00244 +MOVJ EC00244
SMOVL C00245 +MOVJ EC00245
SMOVL C00246 +MOVJ EC00246
SMOVL C00247 +MOVJ EC00247
SMOVL C00248 +MOVJ EC00248
SMOVL C00249 +MOVJ EC00249
SMOVL C00250 +MOVJ EC00250
SMOVL C00251 +MOVJ EC00251
SMOVL C00252 +MOVJ EC00252
SMOVL C00253 +MOVJ EC00253
SMOVL C00254 +MOVJ EC00254
SMOVL C00255 +MOVJ EC00255
SMOVL C00256 +MOVJ EC00256
SMOVL C00257 +MOVJ EC00257
SMOVL C00258 +MOVJ EC00258
SMOVL C00259 +MOVJ EC00259
SMOVL C00260 +MOVJ EC00260
SMOVL C00261 +MOVJ EC00261
SMOVL C00262 +MOVJ EC00262
SMOVL C00263 +MOVJ EC00263
SMOVL C00264 +MOVJ EC00264
SMOVL C00265 +MOVJ EC00265
SMOVL C00266 +MOVJ EC00266
SMOVL C00267 +MOVJ EC00267
SMOVL C00268 +MOVJ EC00268
SMOVL C00269 +MOVJ EC00269
SMOVL C00270 +MOVJ EC00270
SMOVL C00271 +MOVJ EC00271
SMOVL C00272 +MOVJ EC00272
SMOVL C00273 +MOVJ EC00273
SMOVL C00274 +MOVJ EC00274
SMOVL C00275 +MOVJ EC00275
SMOVL C00276 +MOVJ EC00276
SMOVL C00277 +MOVJ EC00277
SMOVL C00278 +MOVJ EC00278
SMOVL C00279 +MOVJ EC00279
SMOVL C00280 +MOVJ EC00280
SMOVL C00281 +MOVJ EC00281
SMOVL C00282 +MOVJ EC00282
SMOVL C00283 +MOVJ EC00283
SMOVL C00284 +MOVJ EC00284
SMOVL C00285 +MOVJ EC00285
SMOVL C00286 +MOVJ EC00286
SMOVL C00287 +MOVJ EC00287
SMOVL C00288 +MOVJ EC00288
SMOVL C00289 +MOVJ EC00289
SMOVL C00290 +MOVJ EC00290
SMOVL C00291 +MOVJ EC00291
SMOVL C00292 +MOVJ EC00292
SMOVL C00293 +MOVJ EC00293
SMOVL C00294 +MOVJ EC00294
SMOVL C00295 +MOVJ EC00295
SMOVL C00296 +MOVJ EC00296
SMOVL C00297 +MOVJ EC00297
SMOVL C00298 +MOVJ EC00298
SMOVL C00299 +MOVJ EC00299
SMOVL C00300 +MOVJ EC00300
SMOVL C00301 +MOVJ EC00301
SMOVL C00302 +MOVJ EC00302
SMOVL C00303 +MOVJ EC00303
SMOVL C00304 +MOVJ EC00304
SMOVL C00305 +MOVJ EC00305
SMOVL C00306 +MOVJ EC00306
SMOVL C00307 +MOVJ EC00307
SMOVL C00308 +MOVJ EC00308
SMOVL C00309 +MOVJ EC00309
SMOVL C00310 +MOVJ EC00310
SMOVL C00311 +MOVJ EC00311
SMOVL C00312 +MOVJ EC00312
SMOVL C00313 +MOVJ EC00313
SMOVL C00314 +MOVJ EC00314
SMOVL C00315 +MOVJ EC00315
SMOVL C00316 +MOVJ EC00316
SMOVL C00317 +MOVJ EC00317
SMOVL C00318 +MOVJ EC00318
SMOVL C00319 +MOVJ EC00319
SMOVL C00320 +MOVJ EC00320
SMOVL C00321 +MOVJ EC00321
SMOVL C00322 +MOVJ EC00322
SMOVL C00323 +MOVJ EC00323
SMOVL C00324 +MOVJ EC00324
SMOVL C00325 +MOVJ EC00325
SMOVL C00326 +MOVJ EC00326
SMOVL C00327 +MOVJ EC00327
SMOVL C00328 +MOVJ EC00328
SMOVL C00329 +MOVJ EC00329
SMOVL C00330 +MOVJ EC00330
SMOVL C00331 +MOVJ EC00331
SMOVL C00332 +MOVJ EC00332
SMOVL C00333 +MOVJ EC00333
SMOVL C00334 +MOVJ EC00334
SMOVL C00335 +MOVJ EC00335
SMOVL C00336 +MOVJ EC00336
SMOVL C00337 +MOVJ EC00337
SMOVL C00338 +MOVJ EC00338
SMOVL C00339 +MOVJ EC00339
SMOVL C00340 +MOVJ EC00340
SMOVL C00341 +MOVJ EC00341
SMOVL C00342 +MOVJ EC00342
SMOVL C00343 +MOVJ EC00343
SMOVL C00344 +MOVJ EC00344
SMOVL C00345 +MOVJ EC00345
SMOVL C00346 +MOVJ EC00346
SMOVL C00347 +MOVJ EC00347
SMOVL C00348 +MOVJ EC00348
SMOVL C00349 +MOVJ EC00349
SMOVL C00350 +MOVJ EC00350
SMOVL C00351 +MOVJ EC00351
SMOVL C00352 +MOVJ EC00352
SMOVL C00353 +MOVJ EC00353
SMOVL C00354 +MOVJ EC00354
SMOVL C00355 +MOVJ EC00355
SMOVL C00356 +MOVJ EC00356
SMOVL C00357 +MOVJ EC00357
SMOVL C00358 +MOVJ EC00358
SMOVL C00359 +MOVJ EC00359
SMOVL C00360 +MOVJ EC00360
SMOVL C00361 +MOVJ EC00361
SMOVL C00362 +MOVJ EC00362
SMOVL C00363 +MOVJ EC00363
SMOVL C00364 +MOVJ EC00364
SMOVL C00365 +MOVJ EC00365
SMOVL C00366 +MOVJ EC00366
SMOVL C00367 +MOVJ EC00367
SMOVL C00368 +MOVJ EC00368
SMOVL C00369 +MOVJ EC00369
SMOVL C00370 +MOVJ EC00370
SMOVL C00371 +MOVJ EC00371
SMOVL C00372 +MOVJ EC00372
SMOVL C00373 +MOVJ EC00373
SMOVL C00374 +MOVJ EC00374
SMOVL C00375 +MOVJ EC00375
SMOVL C00376 +MOVJ EC00376
SMOVL C00377 +MOVJ EC00377
SMOVL C00378 +MOVJ EC00378
SMOVL C00379 +MOVJ EC00379
SMOVL C00380 +MOVJ EC00380
SMOVL C00381 +MOVJ EC00381
SMOVL C00382 +MOVJ EC00382
SMOVL C00383 +MOVJ EC00383
SMOVL C00384 +MOVJ EC00384
SMOVL C00385 +MOVJ EC00385
SMOVL C00386 +MOVJ EC00386
SMOVL C00387 +MOVJ EC00387
SMOVL C00388 +MOVJ EC00388
SMOVL C00389 +MOVJ EC00389
SMOVL C00390 +MOVJ EC00390
SMOVL C00391 +MOVJ EC00391
SMOVL C00392 +MOVJ EC00392
SMOVL C00393 +MOVJ EC00393
SMOVL C00394 +MOVJ EC00394
SMOVL C00395 +MOVJ EC00395
SMOVL C00396 +MOVJ EC00396
SMOVL C00397 +MOVJ EC00397
SMOVL C00398 +MOVJ EC00398
SMOVL C00399 +MOVJ EC00399
SMOVL C00400 +MOVJ EC00400
SMOVL C00401 +MOVJ EC00401
SMOVL C00402 +MOVJ EC00402
SMOVL C00403 +MOVJ EC00403
SMOVL C00404 +MOVJ EC00404
SMOVL C00405 +MOVJ EC00405
SMOVL C00406 +MOVJ EC00406
SMOVL C00407 +MOVJ EC00407
SMOVL C00408 +MOVJ EC00408
SMOVL C00409 +MOVJ EC00409
SMOVL C00410 +MOVJ EC00410
SMOVL C00411 +MOVJ EC00411
SMOVL C00412 +MOVJ EC00412
SMOVL C00413 +MOVJ EC00413
SMOVL C00414 +MOVJ EC00414
SMOVL C00415 +MOVJ EC00415
SMOVL C00416 +MOVJ EC00416
SMOVL C00417 +MOVJ EC00417
SMOVL C00418 +MOVJ EC00418
SMOVL C00419 +MOVJ EC00419
SMOVL C00420 +MOVJ EC00420
SMOVL C00421 +MOVJ EC00421
SMOVL C00422 +MOVJ EC00422
SMOVL C00423 +MOVJ EC00423
SMOVL C00424 +MOVJ EC00424
SMOVL C00425 +MOVJ EC00425
SMOVL C00426 +MOVJ EC00426
SMOVL C00427 +MOVJ EC00427
SMOVL C00428 +MOVJ EC00428
SMOVL C00429 +MOVJ EC00429
SMOVL C00430 +MOVJ EC00430
SMOVL C00431 +MOVJ EC00431
SMOVL C00432 +MOVJ EC00432
SMOVL C00433 +MOVJ EC00433
SMOVL C00434 +MOVJ EC00434
SMOVL C00435 +MOVJ EC00435
SMOVL C00436 +MOVJ EC00436
SMOVL C00437 +MOVJ EC00437
SMOVL C00438 +MOVJ EC00438
SMOVL C00439 +MOVJ EC00439
SMOVL C00440 +MOVJ EC00440
SMOVL C00441 +MOVJ EC00441
SMOVL C00442 +MOVJ EC00442
SMOVL C00443 +MOVJ EC00443
SMOVL C00444 +MOVJ EC00444
SMOVL C00445 +MOVJ EC00445
SMOVL C00446 +MOVJ EC00446
SMOVL C00447 +MOVJ EC00447
SMOVL C00448 +MOVJ EC00448
SMOVL C00449 +MOVJ EC00449
SMOVL C00450 +MOVJ EC00450
SMOVL C00451 +MOVJ EC00451
SMOVL C00452 +MOVJ EC00452
SMOVL C00453 +MOVJ EC00453
SMOVL C00454 +MOVJ EC00454
SMOVL C00455 +MOVJ EC00455
SMOVL C00456 +MOVJ EC00456
SMOVL C00457 +MOVJ EC00457
SMOVL C00458 +MOVJ EC00458
SMOVL C00459 +MOVJ EC00459
SMOVL C00460 +MOVJ EC00460
SMOVL C00461 +MOVJ EC00461
SMOVL C00462 +MOVJ EC00462
SMOVL C00463 +MOVJ EC00463
SMOVL C00464 +MOVJ EC00464
SMOVL C00465 +MOVJ EC00465
SMOVL C00466 +MOVJ EC00466
SMOVL C00467 +MOVJ EC00467
SMOVL C00468 +MOVJ EC00468
SMOVL C00469 +MOVJ EC00469
SMOVL C00470 +MOVJ EC00470
SMOVL C00471 +MOVJ EC00471
SMOVL C00472 +MOVJ EC00472
SMOVL C00473 +MOVJ EC00473
SMOVL C00474 +MOVJ EC00474
SMOVL C00475 +MOVJ EC00475
SMOVL C00476 +MOVJ EC00476
SMOVL C00477 +MOVJ EC00477
SMOVL C00478 +MOVJ EC00478
SMOVL C00479 +MOVJ EC00479
SMOVL C00480 +MOVJ EC00480
SMOVL C00481 +MOVJ EC00481
SMOVL C00482 +MOVJ EC00482
SMOVL C00483 +MOVJ EC00483
SMOVL C00484 +MOVJ EC00484
SMOVL C00485 +MOVJ EC00485
SMOVL C00486 +MOVJ EC00486
SMOVL C00487 +MOVJ EC00487
SMOVL C00488 +MOVJ EC00488
SMOVL C00489 +MOVJ EC00489
SMOVL C00490 +MOVJ EC00490
SMOVL C00491 +MOVJ EC00491
SMOVL C00492 +MOVJ EC00492
SMOVL C00493 +MOVJ EC00493
SMOVL C00494 +MOVJ EC00494
SMOVL C00495 +MOVJ EC00495
SMOVL C00496 +MOVJ EC00496
SMOVL C00497 +MOVJ EC00497
SMOVL C00498 +MOVJ EC00498
SMOVL C00499 +MOVJ EC00499
SMOVL C00500 +MOVJ EC00500
SMOVL C00501 +MOVJ EC00501
SMOVL C00502 +MOVJ EC00502
SMOVL C00503 +MOVJ EC00503
SMOVL C00504 +MOVJ EC00504
SMOVL C00505 +MOVJ EC00505
SMOVL C00506 +MOVJ EC00506
SMOVL C00507 +MOVJ EC00507
SMOVL C00508 +MOVJ EC00508
SMOVL C00509 +MOVJ EC00509
SMOVL C00510 +MOVJ EC00510
SMOVL C00511 +MOVJ EC00511
SMOVL C00512 +MOVJ EC00512
SMOVL C00513 +MOVJ EC00513
SMOVL C00514 +MOVJ EC00514
SMOVL C00515 +MOVJ EC00515
SMOVL C00516 +MOVJ EC00516
SMOVL C00517 +MOVJ EC00517
SMOVL C00518 +MOVJ EC00518
SMOVL C00519 +MOVJ EC00519
SMOVL C00520 +MOVJ EC00520
SMOVL C00521 +MOVJ EC00521
SMOVL C00522 +MOVJ EC00522
SMOVL C00523 +MOVJ EC00523
SMOVL C00524 +MOVJ EC00524
SMOVL C00525 +MOVJ EC00525
SMOVL C00526 +MOVJ EC00526
SMOVL C00527 +MOVJ EC00527
SMOVL C00528 +MOVJ EC00528
SMOVL C00529 +MOVJ EC00529
SMOVL C00530 +MOVJ EC00530
SMOVL C00531 +MOVJ EC00531
SMOVL C00532 +MOVJ EC00532
SMOVL C00533 +MOVJ EC00533
SMOVL C00534 +MOVJ EC00534
SMOVL C00535 +MOVJ EC00535
SMOVL C00536 +MOVJ EC00536
SMOVL C00537 +MOVJ EC00537
SMOVL C00538 +MOVJ EC00538
SMOVL C00539 +MOVJ EC00539
SMOVL C00540 +MOVJ EC00540
SMOVL C00541 +MOVJ EC00541
SMOVL C00542 +MOVJ EC00542
SMOVL C00543 +MOVJ EC00543
SMOVL C00544 +MOVJ EC00544
SMOVL C00545 +MOVJ EC00545
SMOVL C00546 +MOVJ EC00546
SMOVL C00547 +MOVJ EC00547
SMOVL C00548 +MOVJ EC00548
SMOVL C00549 +MOVJ EC00549
SMOVL C00550 +MOVJ EC00550
SMOVL C00551 +MOVJ EC00551
SMOVL C00552 +MOVJ EC00552
SMOVL C00553 +MOVJ EC00553
SMOVL C00554 +MOVJ EC00554
SMOVL C00555 +MOVJ EC00555
SMOVL C00556 +MOVJ EC00556
SMOVL C00557 +MOVJ EC00557
SMOVL C00558 +MOVJ EC00558
SMOVL C00559 +MOVJ EC00559
SMOVL C00560 +MOVJ EC00560
SMOVL C00561 +MOVJ EC00561
SMOVL C00562 +MOVJ EC00562
SMOVL C00563 +MOVJ EC00563
SMOVL C00564 +MOVJ EC00564
SMOVL C00565 +MOVJ EC00565
SMOVL C00566 +MOVJ EC00566
SMOVL C00567 +MOVJ EC00567
SMOVL C00568 +MOVJ EC00568
SMOVL C00569 +MOVJ EC00569
SMOVL C00570 +MOVJ EC00570
SMOVL C00571 +MOVJ EC00571
SMOVL C00572 +MOVJ EC00572
SMOVL C00573 +MOVJ EC00573
SMOVL C00574 +MOVJ EC00574
SMOVL C00575 +MOVJ EC00575
SMOVL C00576 +MOVJ EC00576
SMOVL C00577 +MOVJ EC00577
SMOVL C00578 +MOVJ EC00578
SMOVL C00579 +MOVJ EC00579
SMOVL C00580 +MOVJ EC00580
SMOVL C00581 +MOVJ EC00581
SMOVL C00582 +MOVJ EC00582
SMOVL C00583 +MOVJ EC00583
SMOVL C00584 +MOVJ EC00584
SMOVL C00585 +MOVJ EC00585
SMOVL C00586 +MOVJ EC00586
SMOVL C00587 +MOVJ EC00587
SMOVL C00588 +MOVJ EC00588
SMOVL C00589 +MOVJ EC00589
SMOVL C00590 +MOVJ EC00590
SMOVL C00591 +MOVJ EC00591
SMOVL C00592 +MOVJ EC00592
SMOVL C00593 +MOVJ EC00593
SMOVL C00594 +MOVJ EC00594
SMOVL C00595 +MOVJ EC00595
SMOVL C00596 +MOVJ EC00596
SMOVL C00597 +MOVJ EC00597
SMOVL C00598 +MOVJ EC00598
SMOVL C00599 +MOVJ EC00599
SMOVL C00600 +MOVJ EC00600
SMOVL C00601 +MOVJ EC00601
SMOVL C00602 +MOVJ EC00602
SMOVL C00603 +MOVJ EC00603
SMOVL C00604 +MOVJ EC00604
SMOVL C00605 +MOVJ EC00605
SMOVL C00606 +MOVJ EC00606
SMOVL C00607 +MOVJ EC00607
SMOVL C00608 +MOVJ EC00608
SMOVL C00609 +MOVJ EC00609
SMOVL C00610 +MOVJ EC00610
SMOVL C00611 +MOVJ EC00611
SMOVL C00612 +MOVJ EC00612
SMOVL C00613 +MOVJ EC00613
SMOVL C00614 +MOVJ EC00614
SMOVL C00615 +MOVJ EC00615
SMOVL C00616 +MOVJ EC00616
SMOVL C00617 +MOVJ EC00617
SMOVL C00618 +MOVJ EC00618
SMOVL C00619 +MOVJ EC00619
SMOVL C00620 +MOVJ EC00620
SMOVL C00621 +MOVJ EC00621
SMOVL C00622 +MOVJ EC00622
SMOVL C00623 +MOVJ EC00623
SMOVL C00624 +MOVJ EC00624
SMOVL C00625 +MOVJ EC00625
SMOVL C00626 +MOVJ EC00626
SMOVL C00627 +MOVJ EC00627
SMOVL C00628 +MOVJ EC00628
SMOVL C00629 +MOVJ EC00629
SMOVL C00630 +MOVJ EC00630
SMOVL C00631 +MOVJ EC00631
SMOVL C00632 +MOVJ EC00632
SMOVL C00633 +MOVJ EC00633
SMOVL C00634 +MOVJ EC00634
SMOVL C00635 +MOVJ EC00635
SMOVL C00636 +MOVJ EC00636
SMOVL C00637 +MOVJ EC00637
SMOVL C00638 +MOVJ EC00638
SMOVL C00639 +MOVJ EC00639
SMOVL C00640 +MOVJ EC00640
SMOVL C00641 +MOVJ EC00641
SMOVL C00642 +MOVJ EC00642
SMOVL C00643 +MOVJ EC00643
SMOVL C00644 +MOVJ EC00644
SMOVL C00645 +MOVJ EC00645
SMOVL C00646 +MOVJ EC00646
SMOVL C00647 +MOVJ EC00647
SMOVL C00648 +MOVJ EC00648
SMOVL C00649 +MOVJ EC00649
SMOVL C00650 +MOVJ EC00650
SMOVL C00651 +MOVJ EC00651
SMOVL C00652 +MOVJ EC00652
SMOVL C00653 +MOVJ EC00653
SMOVL C00654 +MOVJ EC00654
SMOVL C00655 +MOVJ EC00655
SMOVL C00656 +MOVJ EC00656
SMOVL C00657 +MOVJ EC00657
SMOVL C00658 +MOVJ EC00658
SMOVL C00659 +MOVJ EC00659
SMOVL C00660 +MOVJ EC00660
SMOVL C00661 +MOVJ EC00661
SMOVL C00662 +MOVJ EC00662
SMOVL C00663 +MOVJ EC00663
SMOVL C00664 +MOVJ EC00664
SMOVL C00665 +MOVJ EC00665
SMOVL C00666 +MOVJ EC00666
SMOVL C00667 +MOVJ EC00667
SMOVL C00668 +MOVJ EC00668
SMOVL C00669 +MOVJ EC00669
SMOVL C00670 +MOVJ EC00670
SMOVL C00671 +MOVJ EC00671
SMOVL C00672 +MOVJ EC00672
SMOVL C00673 +MOVJ EC00673
SMOVL C00674 +MOVJ EC00674
SMOVL C00675 +MOVJ EC00675
SMOVL C00676 +MOVJ EC00676
SMOVL C00677 +MOVJ EC00677
SMOVL C00678 +MOVJ EC00678
SMOVL C00679 +MOVJ EC00679
SMOVL C00680 +MOVJ EC00680
SMOVL C00681 +MOVJ EC00681
SMOVL C00682 +MOVJ EC00682
SMOVL C00683 +MOVJ EC00683
SMOVL C00684 +MOVJ EC00684
SMOVL C00685 +MOVJ EC00685
SMOVL C00686 +MOVJ EC00686
SMOVL C00687 +MOVJ EC00687
SMOVL C00688 +MOVJ EC00688
SMOVL C00689 +MOVJ EC00689
SMOVL C00690 +MOVJ EC00690
SMOVL C00691 +MOVJ EC00691
SMOVL C00692 +MOVJ EC00692
SMOVL C00693 +MOVJ EC00693
SMOVL C00694 +MOVJ EC00694
SMOVL C00695 +MOVJ EC00695
SMOVL C00696 +MOVJ EC00696
SMOVL C00697 +MOVJ EC00697
SMOVL C00698 +MOVJ EC00698
SMOVL C00699 +MOVJ EC00699
SMOVL C00700 +MOVJ EC00700
SMOVL C00701 +MOVJ EC00701
SMOVL C00702 +MOVJ EC00702
SMOVL C00703 +MOVJ EC00703
SMOVL C00704 +MOVJ EC00704
SMOVL C00705 +MOVJ EC00705
SMOVL C00706 +MOVJ EC00706
SMOVL C00707 +MOVJ EC00707
SMOVL C00708 +MOVJ EC00708
SMOVL C00709 +MOVJ EC00709
SMOVL C00710 +MOVJ EC00710
SMOVL C00711 +MOVJ EC00711
SMOVL C00712 +MOVJ EC00712
SMOVL C00713 +MOVJ EC00713
SMOVL C00714 +MOVJ EC00714
SMOVL C00715 +MOVJ EC00715
SMOVL C00716 +MOVJ EC00716
SMOVL C00717 +MOVJ EC00717
SMOVL C00718 +MOVJ EC00718
SMOVL C00719 +MOVJ EC00719
SMOVL C00720 +MOVJ EC00720
SMOVL C00721 +MOVJ EC00721
SMOVL C00722 +MOVJ EC00722
SMOVL C00723 +MOVJ EC00723
SMOVL C00724 +MOVJ EC00724
SMOVL C00725 +MOVJ EC00725
SMOVL C00726 +MOVJ EC00726
SMOVL C00727 +MOVJ EC00727
SMOVL C00728 +MOVJ EC00728
SMOVL C00729 +MOVJ EC00729
SMOVL C00730 +MOVJ EC00730
SMOVL C00731 +MOVJ EC00731
SMOVL C00732 +MOVJ EC00732
SMOVL C00733 +MOVJ EC00733
SMOVL C00734 +MOVJ EC00734
SMOVL C00735 +MOVJ EC00735
SMOVL C00736 +MOVJ EC00736
SMOVL C00737 +MOVJ EC00737
SMOVL C00738 +MOVJ EC00738
SMOVL C00739 +MOVJ EC00739
SMOVL C00740 +MOVJ EC00740
SMOVL C00741 +MOVJ EC00741
SMOVL C00742 +MOVJ EC00742
SMOVL C00743 +MOVJ EC00743
SMOVL C00744 +MOVJ EC00744
SMOVL C00745 +MOVJ EC00745
SMOVL C00746 +MOVJ EC00746
SMOVL C00747 +MOVJ EC00747
SMOVL C00748 +MOVJ EC00748
SMOVL C00749 +MOVJ EC00749
SMOVL C00750 +MOVJ EC00750
SMOVL C00751 +MOVJ EC00751
SMOVL C00752 +MOVJ EC00752
SMOVL C00753 +MOVJ EC00753
SMOVL C00754 +MOVJ EC00754
SMOVL C00755 +MOVJ EC00755
SMOVL C00756 +MOVJ EC00756
SMOVL C00757 +MOVJ EC00757
SMOVL C00758 +MOVJ EC00758
SMOVL C00759 +MOVJ EC00759
SMOVL C00760 +MOVJ EC00760
SMOVL C00761 +MOVJ EC00761
SMOVL C00762 +MOVJ EC00762
SMOVL C00763 +MOVJ EC00763
SMOVL C00764 +MOVJ EC00764
SMOVL C00765 +MOVJ EC00765
SMOVL C00766 +MOVJ EC00766
SMOVL C00767 +MOVJ EC00767
SMOVL C00768 +MOVJ EC00768
SMOVL C00769 +MOVJ EC00769
SMOVL C00770 +MOVJ EC00770
SMOVL C00771 +MOVJ EC00771
SMOVL C00772 +MOVJ EC00772
SMOVL C00773 +MOVJ EC00773
SMOVL C00774 +MOVJ EC00774
SMOVL C00775 +MOVJ EC00775
SMOVL C00776 +MOVJ EC00776
SMOVL C00777 +MOVJ EC00777
SMOVL C00778 +MOVJ EC00778
SMOVL C00779 +MOVJ EC00779
SMOVL C00780 +MOVJ EC00780
SMOVL C00781 +MOVJ EC00781
SMOVL C00782 +MOVJ EC00782
SMOVL C00783 +MOVJ EC00783
SMOVL C00784 +MOVJ EC00784
SMOVL C00785 +MOVJ EC00785
SMOVL C00786 +MOVJ EC00786
SMOVL C00787 +MOVJ EC00787
SMOVL C00788 +MOVJ EC00788
SMOVL C00789 +MOVJ EC00789
SMOVL C00790 +MOVJ EC00790
SMOVL C00791 +MOVJ EC00791
SMOVL C00792 +MOVJ EC00792
SMOVL C00793 +MOVJ EC00793
SMOVL C00794 +MOVJ EC00794
SMOVL C00795 +MOVJ EC00795
SMOVL C00796 +MOVJ EC00796
SMOVL C00797 +MOVJ EC00797
SMOVL C00798 +MOVJ EC00798
SMOVL C00799 +MOVJ EC00799
SMOVL C00800 +MOVJ EC00800
SMOVL C00801 +MOVJ EC00801
SMOVL C00802 +MOVJ EC00802
SMOVL C00803 +MOVJ EC00803
SMOVL C00804 +MOVJ EC00804
SMOVL C00805 +MOVJ EC00805
SMOVL C00806 +MOVJ EC00806
SMOVL C00807 +MOVJ EC00807
SMOVL C00808 +MOVJ EC00808
SMOVL C00809 +MOVJ EC00809
SMOVL C00810 +MOVJ EC00810
SMOVL C00811 +MOVJ EC00811
SMOVL C00812 +MOVJ EC00812
SMOVL C00813 +MOVJ EC00813
SMOVL C00814 +MOVJ EC00814
SMOVL C00815 +MOVJ EC00815
SMOVL C00816 +MOVJ EC00816
SMOVL C00817 +MOVJ EC00817
SMOVL C00818 +MOVJ EC00818
SMOVL C00819 +MOVJ EC00819
SMOVL C00820 +MOVJ EC00820
SMOVL C00821 +MOVJ EC00821
SMOVL C00822 +MOVJ EC00822
SMOVL C00823 +MOVJ EC00823
SMOVL C00824 +MOVJ EC00824
SMOVL C00825 +MOVJ EC00825
SMOVL C00826 +MOVJ EC00826
SMOVL C00827 +MOVJ EC00827
SMOVL C00828 +MOVJ EC00828
SMOVL C00829 +MOVJ EC00829
SMOVL C00830 +MOVJ EC00830
SMOVL C00831 +MOVJ EC00831
SMOVL C00832 +MOVJ EC00832
SMOVL C00833 +MOVJ EC00833
SMOVL C00834 +MOVJ EC00834
SMOVL C00835 +MOVJ EC00835
SMOVL C00836 +MOVJ EC00836
SMOVL C00837 +MOVJ EC00837
SMOVL C00838 +MOVJ EC00838
SMOVL C00839 +MOVJ EC00839
SMOVL C00840 +MOVJ EC00840
SMOVL C00841 +MOVJ EC00841
SMOVL C00842 +MOVJ EC00842
SMOVL C00843 +MOVJ EC00843
SMOVL C00844 +MOVJ EC00844
SMOVL C00845 +MOVJ EC00845
SMOVL C00846 +MOVJ EC00846
SMOVL C00847 +MOVJ EC00847
SMOVL C00848 +MOVJ EC00848
SMOVL C00849 +MOVJ EC00849
SMOVL C00850 +MOVJ EC00850
SMOVL C00851 +MOVJ EC00851
SMOVL C00852 +MOVJ EC00852
SMOVL C00853 +MOVJ EC00853
SMOVL C00854 +MOVJ EC00854
SMOVL C00855 +MOVJ EC00855
SMOVL C00856 +MOVJ EC00856
SMOVL C00857 +MOVJ EC00857
SMOVL C00858 +MOVJ EC00858
SMOVL C00859 +MOVJ EC00859
SMOVL C00860 +MOVJ EC00860
SMOVL C00861 +MOVJ EC00861
SMOVL C00862 +MOVJ EC00862
SMOVL C00863 +MOVJ EC00863
SMOVL C00864 +MOVJ EC00864
SMOVL C00865 +MOVJ EC00865
SMOVL C00866 +MOVJ EC00866
SMOVL C00867 +MOVJ EC00867
SMOVL C00868 +MOVJ EC00868
SMOVL C00869 +MOVJ EC00869
SMOVL C00870 +MOVJ EC00870
SMOVL C00871 +MOVJ EC00871
SMOVL C00872 +MOVJ EC00872
SMOVL C00873 +MOVJ EC00873
SMOVL C00874 +MOVJ EC00874
SMOVL C00875 +MOVJ EC00875
SMOVL C00876 +MOVJ EC00876
SMOVL C00877 +MOVJ EC00877
SMOVL C00878 +MOVJ EC00878
SMOVL C00879 +MOVJ EC00879
SMOVL C00880 +MOVJ EC00880
SMOVL C00881 +MOVJ EC00881
SMOVL C00882 +MOVJ EC00882
SMOVL C00883 +MOVJ EC00883
SMOVL C00884 +MOVJ EC00884
SMOVL C00885 +MOVJ EC00885
SMOVL C00886 +MOVJ EC00886
SMOVL C00887 +MOVJ EC00887
SMOVL C00888 +MOVJ EC00888
SMOVL C00889 +MOVJ EC00889
SMOVL C00890 +MOVJ EC00890
SMOVL C00891 +MOVJ EC00891
SMOVL C00892 +MOVJ EC00892
SMOVL C00893 +MOVJ EC00893
SMOVL C00894 +MOVJ EC00894
SMOVL C00895 +MOVJ EC00895
SMOVL C00896 +MOVJ EC00896
SMOVL C00897 +MOVJ EC00897
SMOVL C00898 +MOVJ EC00898
SMOVL C00899 +MOVJ EC00899
SMOVL C00900 +MOVJ EC00900
SMOVL C00901 +MOVJ EC00901
SMOVL C00902 +MOVJ EC00902
SMOVL C00903 +MOVJ EC00903
SMOVL C00904 +MOVJ EC00904
SMOVL C00905 +MOVJ EC00905
SMOVL C00906 +MOVJ EC00906
SMOVL C00907 +MOVJ EC00907
SMOVL C00908 +MOVJ EC00908
SMOVL C00909 +MOVJ EC00909
SMOVL C00910 +MOVJ EC00910
SMOVL C00911 +MOVJ EC00911
SMOVL C00912 +MOVJ EC00912
SMOVL C00913 +MOVJ EC00913
SMOVL C00914 +MOVJ EC00914
SMOVL C00915 +MOVJ EC00915
SMOVL C00916 +MOVJ EC00916
SMOVL C00917 +MOVJ EC00917
SMOVL C00918 +MOVJ EC00918
SMOVL C00919 +MOVJ EC00919
SMOVL C00920 +MOVJ EC00920
SMOVL C00921 +MOVJ EC00921
SMOVL C00922 +MOVJ EC00922
SMOVL C00923 +MOVJ EC00923
SMOVL C00924 +MOVJ EC00924
SMOVL C00925 +MOVJ EC00925
SMOVL C00926 +MOVJ EC00926
SMOVL C00927 +MOVJ EC00927
SMOVL C00928 +MOVJ EC00928
SMOVL C00929 +MOVJ EC00929
SMOVL C00930 +MOVJ EC00930
SMOVL C00931 +MOVJ EC00931
SMOVL C00932 +MOVJ EC00932
SMOVL C00933 +MOVJ EC00933
SMOVL C00934 +MOVJ EC00934
SMOVL C00935 +MOVJ EC00935
SMOVL C00936 +MOVJ EC00936
SMOVL C00937 +MOVJ EC00937
SMOVL C00938 +MOVJ EC00938
SMOVL C00939 +MOVJ EC00939
SMOVL C00940 +MOVJ EC00940
SMOVL C00941 +MOVJ EC00941
SMOVL C00942 +MOVJ EC00942
SMOVL C00943 +MOVJ EC00943
SMOVL C00944 +MOVJ EC00944
SMOVL C00945 +MOVJ EC00945
SMOVL C00946 +MOVJ EC00946
SMOVL C00947 +MOVJ EC00947
SMOVL C00948 +MOVJ EC00948
SMOVL C00949 +MOVJ EC00949
SMOVL C00950 +MOVJ EC00950
SMOVL C00951 +MOVJ EC00951
SMOVL C00952 +MOVJ EC00952
SMOVL C00953 +MOVJ EC00953
SMOVL C00954 +MOVJ EC00954
SMOVL C00955 +MOVJ EC00955
SMOVL C00956 +MOVJ EC00956
SMOVL C00957 +MOVJ EC00957
SMOVL C00958 +MOVJ EC00958
SMOVL C00959 +MOVJ EC00959
SMOVL C00960 +MOVJ EC00960
SMOVL C00961 +MOVJ EC00961
SMOVL C00962 +MOVJ EC00962
SMOVL C00963 +MOVJ EC00963
SMOVL C00964 +MOVJ EC00964
SMOVL C00965 +MOVJ EC00965
SMOVL C00966 +MOVJ EC00966
SMOVL C00967 +MOVJ EC00967
SMOVL C00968 +MOVJ EC00968
SMOVL C00969 +MOVJ EC00969
SMOVL C00970 +MOVJ EC00970
SMOVL C00971 +MOVJ EC00971
SMOVL C00972 +MOVJ EC00972
SMOVL C00973 +MOVJ EC00973
SMOVL C00974 +MOVJ EC00974
SMOVL C00975 +MOVJ EC00975
SMOVL C00976 +MOVJ EC00976
SMOVL C00977 +MOVJ EC00977
SMOVL C00978 +MOVJ EC00978
SMOVL C00979 +MOVJ EC00979
SMOVL C00980 +MOVJ EC00980
SMOVL C00981 +MOVJ EC00981
SMOVL C00982 +MOVJ EC00982
SMOVL C00983 +MOVJ EC00983
SMOVL C00984 +MOVJ EC00984
SMOVL C00985 +MOVJ EC00985
SMOVL C00986 +MOVJ EC00986
SMOVL C00987 +MOVJ EC00987
SMOVL C00988 +MOVJ EC00988
SMOVL C00989 +MOVJ EC00989
SMOVL C00990 +MOVJ EC00990
SMOVL C00991 +MOVJ EC00991
SMOVL C00992 +MOVJ EC00992
SMOVL C00993 +MOVJ EC00993
SMOVL C00994 +MOVJ EC00994
SMOVL C00995 +MOVJ EC00995
SMOVL C00996 +MOVJ EC00996
SMOVL C00997 +MOVJ EC00997
SMOVL C00998 +MOVJ EC00998
SMOVL C00999 +MOVJ EC00999
SMOVL C01000 +MOVJ EC01000
SMOVL C01001 +MOVJ EC01001
SMOVL C01002 +MOVJ EC01002
SMOVL C01003 +MOVJ EC01003
SMOVL C01004 +MOVJ EC01004
SMOVL C01005 +MOVJ EC01005
SMOVL C01006 +MOVJ EC01006
SMOVL C01007 +MOVJ EC01007
SMOVL C01008 +MOVJ EC01008
SMOVL C01009 +MOVJ EC01009
SMOVL C01010 +MOVJ EC01010
SMOVL C01011 +MOVJ EC01011
SMOVL C01012 +MOVJ EC01012
SMOVL C01013 +MOVJ EC01013
SMOVL C01014 +MOVJ EC01014
SMOVL C01015 +MOVJ EC01015
SMOVL C01016 +MOVJ EC01016
SMOVL C01017 +MOVJ EC01017
SMOVL C01018 +MOVJ EC01018
SMOVL C01019 +MOVJ EC01019
SMOVL C01020 +MOVJ EC01020
SMOVL C01021 +MOVJ EC01021
SMOVL C01022 +MOVJ EC01022
SMOVL C01023 +MOVJ EC01023
SMOVL C01024 +MOVJ EC01024
SMOVL C01025 +MOVJ EC01025
SMOVL C01026 +MOVJ EC01026
SMOVL C01027 +MOVJ EC01027
SMOVL C01028 +MOVJ EC01028
SMOVL C01029 +MOVJ EC01029
SMOVL C01030 +MOVJ EC01030
SMOVL C01031 +MOVJ EC01031
SMOVL C01032 +MOVJ EC01032
SMOVL C01033 +MOVJ EC01033
SMOVL C01034 +MOVJ EC01034
SMOVL C01035 +MOVJ EC01035
SMOVL C01036 +MOVJ EC01036
SMOVL C01037 +MOVJ EC01037
SMOVL C01038 +MOVJ EC01038
SMOVL C01039 +MOVJ EC01039
SMOVL C01040 +MOVJ EC01040
SMOVL C01041 +MOVJ EC01041
SMOVL C01042 +MOVJ EC01042
SMOVL C01043 +MOVJ EC01043
SMOVL C01044 +MOVJ EC01044
SMOVL C01045 +MOVJ EC01045
SMOVL C01046 +MOVJ EC01046
SMOVL C01047 +MOVJ EC01047
SMOVL C01048 +MOVJ EC01048
SMOVL C01049 +MOVJ EC01049
SMOVL C01050 +MOVJ EC01050
SMOVL C01051 +MOVJ EC01051
SMOVL C01052 +MOVJ EC01052
SMOVL C01053 +MOVJ EC01053
SMOVL C01054 +MOVJ EC01054
SMOVL C01055 +MOVJ EC01055
SMOVL C01056 +MOVJ EC01056
SMOVL C01057 +MOVJ EC01057
SMOVL C01058 +MOVJ EC01058
SMOVL C01059 +MOVJ EC01059
SMOVL C01060 +MOVJ EC01060
SMOVL C01061 +MOVJ EC01061
SMOVL C01062 +MOVJ EC01062
SMOVL C01063 +MOVJ EC01063
SMOVL C01064 +MOVJ EC01064
SMOVL C01065 +MOVJ EC01065
SMOVL C01066 +MOVJ EC01066
SMOVL C01067 +MOVJ EC01067
SMOVL C01068 +MOVJ EC01068
SMOVL C01069 +MOVJ EC01069
SMOVL C01070 +MOVJ EC01070
SMOVL C01071 +MOVJ EC01071
SMOVL C01072 +MOVJ EC01072
SMOVL C01073 +MOVJ EC01073
SMOVL C01074 +MOVJ EC01074
SMOVL C01075 +MOVJ EC01075
SMOVL C01076 +MOVJ EC01076
SMOVL C01077 +MOVJ EC01077
SMOVL C01078 +MOVJ EC01078
SMOVL C01079 +MOVJ EC01079
SMOVL C01080 +MOVJ EC01080
SMOVL C01081 +MOVJ EC01081
SMOVL C01082 +MOVJ EC01082
SMOVL C01083 +MOVJ EC01083
SMOVL C01084 +MOVJ EC01084
SMOVL C01085 +MOVJ EC01085
SMOVL C01086 +MOVJ EC01086
SMOVL C01087 +MOVJ EC01087
SMOVL C01088 +MOVJ EC01088
SMOVL C01089 +MOVJ EC01089
SMOVL C01090 +MOVJ EC01090
SMOVL C01091 +MOVJ EC01091
SMOVL C01092 +MOVJ EC01092
SMOVL C01093 +MOVJ EC01093
SMOVL C01094 +MOVJ EC01094
SMOVL C01095 +MOVJ EC01095
SMOVL C01096 +MOVJ EC01096
SMOVL C01097 +MOVJ EC01097
SMOVL C01098 +MOVJ EC01098
SMOVL C01099 +MOVJ EC01099
SMOVL C01100 +MOVJ EC01100
SMOVL C01101 +MOVJ EC01101
SMOVL C01102 +MOVJ EC01102
SMOVL C01103 +MOVJ EC01103
SMOVL C01104 +MOVJ EC01104
SMOVL C01105 +MOVJ EC01105
SMOVL C01106 +MOVJ EC01106
SMOVL C01107 +MOVJ EC01107
SMOVL C01108 +MOVJ EC01108
SMOVL C01109 +MOVJ EC01109
SMOVL C01110 +MOVJ EC01110
SMOVL C01111 +MOVJ EC01111
SMOVL C01112 +MOVJ EC01112
SMOVL C01113 +MOVJ EC01113
SMOVL C01114 +MOVJ EC01114
SMOVL C01115 +MOVJ EC01115
SMOVL C01116 +MOVJ EC01116
SMOVL C01117 +MOVJ EC01117
SMOVL C01118 +MOVJ EC01118
SMOVL C01119 +MOVJ EC01119
SMOVL C01120 +MOVJ EC01120
SMOVL C01121 +MOVJ EC01121
SMOVL C01122 +MOVJ EC01122
SMOVL C01123 +MOVJ EC01123
SMOVL C01124 +MOVJ EC01124
SMOVL C01125 +MOVJ EC01125
SMOVL C01126 +MOVJ EC01126
SMOVL C01127 +MOVJ EC01127
SMOVL C01128 +MOVJ EC01128
SMOVL C01129 +MOVJ EC01129
SMOVL C01130 +MOVJ EC01130
SMOVL C01131 +MOVJ EC01131
SMOVL C01132 +MOVJ EC01132
SMOVL C01133 +MOVJ EC01133
SMOVL C01134 +MOVJ EC01134
SMOVL C01135 +MOVJ EC01135
SMOVL C01136 +MOVJ EC01136
SMOVL C01137 +MOVJ EC01137
SMOVL C01138 +MOVJ EC01138
SMOVL C01139 +MOVJ EC01139
SMOVL C01140 +MOVJ EC01140
SMOVL C01141 +MOVJ EC01141
SMOVL C01142 +MOVJ EC01142
SMOVL C01143 +MOVJ EC01143
SMOVL C01144 +MOVJ EC01144
SMOVL C01145 +MOVJ EC01145
SMOVL C01146 +MOVJ EC01146
SMOVL C01147 +MOVJ EC01147
SMOVL C01148 +MOVJ EC01148
SMOVL C01149 +MOVJ EC01149
SMOVL C01150 +MOVJ EC01150
SMOVL C01151 +MOVJ EC01151
SMOVL C01152 +MOVJ EC01152
SMOVL C01153 +MOVJ EC01153
SMOVL C01154 +MOVJ EC01154
SMOVL C01155 +MOVJ EC01155
SMOVL C01156 +MOVJ EC01156
SMOVL C01157 +MOVJ EC01157
SMOVL C01158 +MOVJ EC01158
SMOVL C01159 +MOVJ EC01159
SMOVL C01160 +MOVJ EC01160
SMOVL C01161 +MOVJ EC01161
SMOVL C01162 +MOVJ EC01162
SMOVL C01163 +MOVJ EC01163
SMOVL C01164 +MOVJ EC01164
SMOVL C01165 +MOVJ EC01165
SMOVL C01166 +MOVJ EC01166
SMOVL C01167 +MOVJ EC01167
SMOVL C01168 +MOVJ EC01168
SMOVL C01169 +MOVJ EC01169
SMOVL C01170 +MOVJ EC01170
SMOVL C01171 +MOVJ EC01171
SMOVL C01172 +MOVJ EC01172
SMOVL C01173 +MOVJ EC01173
SMOVL C01174 +MOVJ EC01174
SMOVL C01175 +MOVJ EC01175
SMOVL C01176 +MOVJ EC01176
SMOVL C01177 +MOVJ EC01177
SMOVL C01178 +MOVJ EC01178
SMOVL C01179 +MOVJ EC01179
SMOVL C01180 +MOVJ EC01180
SMOVL C01181 +MOVJ EC01181
SMOVL C01182 +MOVJ EC01182
SMOVL C01183 +MOVJ EC01183
SMOVL C01184 +MOVJ EC01184
SMOVL C01185 +MOVJ EC01185
SMOVL C01186 +MOVJ EC01186
SMOVL C01187 +MOVJ EC01187
SMOVL C01188 +MOVJ EC01188
SMOVL C01189 +MOVJ EC01189
SMOVL C01190 +MOVJ EC01190
SMOVL C01191 +MOVJ EC01191
SMOVL C01192 +MOVJ EC01192
SMOVL C01193 +MOVJ EC01193
SMOVL C01194 +MOVJ EC01194
SMOVL C01195 +MOVJ EC01195
SMOVL C01196 +MOVJ EC01196
SMOVL C01197 +MOVJ EC01197
SMOVL C01198 +MOVJ EC01198
SMOVL C01199 +MOVJ EC01199
SMOVL C01200 +MOVJ EC01200
SMOVL C01201 +MOVJ EC01201
SMOVL C01202 +MOVJ EC01202
SMOVL C01203 +MOVJ EC01203
SMOVL C01204 +MOVJ EC01204
SMOVL C01205 +MOVJ EC01205
SMOVL C01206 +MOVJ EC01206
SMOVL C01207 +MOVJ EC01207
SMOVL C01208 +MOVJ EC01208
SMOVL C01209 +MOVJ EC01209
SMOVL C01210 +MOVJ EC01210
SMOVL C01211 +MOVJ EC01211
SMOVL C01212 +MOVJ EC01212
SMOVL C01213 +MOVJ EC01213
SMOVL C01214 +MOVJ EC01214
SMOVL C01215 +MOVJ EC01215
SMOVL C01216 +MOVJ EC01216
SMOVL C01217 +MOVJ EC01217
SMOVL C01218 +MOVJ EC01218
SMOVL C01219 +MOVJ EC01219
SMOVL C01220 +MOVJ EC01220
SMOVL C01221 +MOVJ EC01221
SMOVL C01222 +MOVJ EC01222
SMOVL C01223 +MOVJ EC01223
SMOVL C01224 +MOVJ EC01224
SMOVL C01225 +MOVJ EC01225
SMOVL C01226 +MOVJ EC01226
SMOVL C01227 +MOVJ EC01227
SMOVL C01228 +MOVJ EC01228
SMOVL C01229 +MOVJ EC01229
SMOVL C01230 +MOVJ EC01230
SMOVL C01231 +MOVJ EC01231
SMOVL C01232 +MOVJ EC01232
SMOVL C01233 +MOVJ EC01233
SMOVL C01234 +MOVJ EC01234
SMOVL C01235 +MOVJ EC01235
SMOVL C01236 +MOVJ EC01236
SMOVL C01237 +MOVJ EC01237
SMOVL C01238 +MOVJ EC01238
SMOVL C01239 +MOVJ EC01239
SMOVL C01240 +MOVJ EC01240
SMOVL C01241 +MOVJ EC01241
SMOVL C01242 +MOVJ EC01242
SMOVL C01243 +MOVJ EC01243
SMOVL C01244 +MOVJ EC01244
SMOVL C01245 +MOVJ EC01245
SMOVL C01246 +MOVJ EC01246
SMOVL C01247 +MOVJ EC01247
SMOVL C01248 +MOVJ EC01248
SMOVL C01249 +MOVJ EC01249
SMOVL C01250 +MOVJ EC01250
SMOVL C01251 +MOVJ EC01251
SMOVL C01252 +MOVJ EC01252
SMOVL C01253 +MOVJ EC01253
SMOVL C01254 +MOVJ EC01254
SMOVL C01255 +MOVJ EC01255
SMOVL C01256 +MOVJ EC01256
SMOVL C01257 +MOVJ EC01257
SMOVL C01258 +MOVJ EC01258
SMOVL C01259 +MOVJ EC01259
SMOVL C01260 +MOVJ EC01260
SMOVL C01261 +MOVJ EC01261
SMOVL C01262 +MOVJ EC01262
SMOVL C01263 +MOVJ EC01263
SMOVL C01264 +MOVJ EC01264
SMOVL C01265 +MOVJ EC01265
SMOVL C01266 +MOVJ EC01266
SMOVL C01267 +MOVJ EC01267
SMOVL C01268 +MOVJ EC01268
SMOVL C01269 +MOVJ EC01269
SMOVL C01270 +MOVJ EC01270
SMOVL C01271 +MOVJ EC01271
SMOVL C01272 +MOVJ EC01272
SMOVL C01273 +MOVJ EC01273
SMOVL C01274 +MOVJ EC01274
SMOVL C01275 +MOVJ EC01275
SMOVL C01276 +MOVJ EC01276
SMOVL C01277 +MOVJ EC01277
SMOVL C01278 +MOVJ EC01278
SMOVL C01279 +MOVJ EC01279
SMOVL C01280 +MOVJ EC01280
SMOVL C01281 +MOVJ EC01281
SMOVL C01282 +MOVJ EC01282
SMOVL C01283 +MOVJ EC01283
SMOVL C01284 +MOVJ EC01284
SMOVL C01285 +MOVJ EC01285
SMOVL C01286 +MOVJ EC01286
SMOVL C01287 +MOVJ EC01287
SMOVL C01288 +MOVJ EC01288
SMOVL C01289 +MOVJ EC01289
SMOVL C01290 +MOVJ EC01290
SMOVL C01291 +MOVJ EC01291
SMOVL C01292 +MOVJ EC01292
SMOVL C01293 +MOVJ EC01293
SMOVL C01294 +MOVJ EC01294
SMOVL C01295 +MOVJ EC01295
SMOVL C01296 +MOVJ EC01296
SMOVL C01297 +MOVJ EC01297
SMOVL C01298 +MOVJ EC01298
SMOVL C01299 +MOVJ EC01299
SMOVL C01300 +MOVJ EC01300
SMOVL C01301 +MOVJ EC01301
SMOVL C01302 +MOVJ EC01302
SMOVL C01303 +MOVJ EC01303
SMOVL C01304 +MOVJ EC01304
SMOVL C01305 +MOVJ EC01305
SMOVL C01306 +MOVJ EC01306
SMOVL C01307 +MOVJ EC01307
SMOVL C01308 +MOVJ EC01308
SMOVL C01309 +MOVJ EC01309
SMOVL C01310 +MOVJ EC01310
SMOVL C01311 +MOVJ EC01311
SMOVL C01312 +MOVJ EC01312
SMOVL C01313 +MOVJ EC01313
SMOVL C01314 +MOVJ EC01314
SMOVL C01315 +MOVJ EC01315
SMOVL C01316 +MOVJ EC01316
SMOVL C01317 +MOVJ EC01317
SMOVL C01318 +MOVJ EC01318
SMOVL C01319 +MOVJ EC01319
SMOVL C01320 +MOVJ EC01320
SMOVL C01321 +MOVJ EC01321
SMOVL C01322 +MOVJ EC01322
SMOVL C01323 +MOVJ EC01323
SMOVL C01324 +MOVJ EC01324
SMOVL C01325 +MOVJ EC01325
SMOVL C01326 +MOVJ EC01326
SMOVL C01327 +MOVJ EC01327
SMOVL C01328 +MOVJ EC01328
SMOVL C01329 +MOVJ EC01329
SMOVL C01330 +MOVJ EC01330
SMOVL C01331 +MOVJ EC01331
SMOVL C01332 +MOVJ EC01332
SMOVL C01333 +MOVJ EC01333
SMOVL C01334 +MOVJ EC01334
SMOVL C01335 +MOVJ EC01335
SMOVL C01336 +MOVJ EC01336
SMOVL C01337 +MOVJ EC01337
SMOVL C01338 +MOVJ EC01338
SMOVL C01339 +MOVJ EC01339
SMOVL C01340 +MOVJ EC01340
SMOVL C01341 +MOVJ EC01341
SMOVL C01342 +MOVJ EC01342
SMOVL C01343 +MOVJ EC01343
SMOVL C01344 +MOVJ EC01344
SMOVL C01345 +MOVJ EC01345
SMOVL C01346 +MOVJ EC01346
SMOVL C01347 +MOVJ EC01347
SMOVL C01348 +MOVJ EC01348
SMOVL C01349 +MOVJ EC01349
SMOVL C01350 +MOVJ EC01350
SMOVL C01351 +MOVJ EC01351
SMOVL C01352 +MOVJ EC01352
SMOVL C01353 +MOVJ EC01353
SMOVL C01354 +MOVJ EC01354
SMOVL C01355 +MOVJ EC01355
SMOVL C01356 +MOVJ EC01356
SMOVL C01357 +MOVJ EC01357
SMOVL C01358 +MOVJ EC01358
SMOVL C01359 +MOVJ EC01359
SMOVL C01360 +MOVJ EC01360
SMOVL C01361 +MOVJ EC01361
SMOVL C01362 +MOVJ EC01362
SMOVL C01363 +MOVJ EC01363
SMOVL C01364 +MOVJ EC01364
SMOVL C01365 +MOVJ EC01365
SMOVL C01366 +MOVJ EC01366
SMOVL C01367 +MOVJ EC01367
SMOVL C01368 +MOVJ EC01368
SMOVL C01369 +MOVJ EC01369
SMOVL C01370 +MOVJ EC01370
SMOVL C01371 +MOVJ EC01371
SMOVL C01372 +MOVJ EC01372
SMOVL C01373 +MOVJ EC01373
